hm 1.12.06		rev 1.2
	corrected failure in sequence logic.
	added init at startup to prevent from initial error after start.

hm 17.1.2007		rev 1.3
	changed output fault to status for better compatibility with other modules (ESR).
	added stop on error functionality and setup variable
	default for inputs in0..3 is true.
	renamed variable state to step

hm	17.sep 2007		rev 1.4
	replaced time() with T_PLC_MS() for compatibility reasons

*)
END_FUNCTION_BLOCK

(* POU Logic/generators/TONOF, ST *)
FUNCTION_BLOCK TONOF
VAR_INPUT
	IN : BOOL;
	T1, T2 : TIME;
END_VAR
VAR_OUTPUT
	Q : BOOL;
END_VAR
VAR
	X : TON;
	Y : TOF;
END_VAR

(*
version 1.1	17 sep 2007
programmer 	hugo
tested by		tobias

TONOF generated a TON and TOF Delay for the Input N TON (T1) and TOF (T2) can be configured separately
*)
X(IN := IN, PT := T1);
Y(in := X.Q, PT := T2);
Q := Y.Q;

(* revision history
hm	10. dec 2007	rev 1.0
	original version

*)
	
END_FUNCTION_BLOCK

(* POU Logic/memory/FIFO_16, ST *)
FUNCTION_BLOCK FIFO_16
VAR_INPUT
	Din : DWORD;
	WR : BOOL;
	E : BOOL;
	RST : BOOL;
END_VAR
VAR_OUTPUT
	Dout : DWORD := 0;
	empty : BOOL := TRUE;
	full : BOOL := FALSE;
END_VAR
VAR
	fifo : ARRAY[0..15] OF DWORD;
	NW : INT := 0;
	NR : INT := 0;
	top : INT := 15;
END_VAR

(*
	version 1.1	19. feb 2008
	programmer 	hugo
	tested by		tobias

16 Dword FIFO memory
*)
IF rst THEN
	(* asynchronous reset for the fifo *)
	NW := 0;
	NR := 0;
	Dout := 0;
	empty := TRUE;
	full := FALSE;
ELSIF WR AND E AND NOT full THEN
	(* write action *)
	fifo[NW] := Din;
	IF NW = top THEN NW := 0; ELSE NW := NW + 1; END_IF;
	full := NW = NR;
	empty := FALSE;
ELSIF NOT WR AND E AND NOT empty THEN
	(* read from stack *)
	Dout := fifo[NR];
	IF NR = top THEN NR := 0; ELSE NR := NR + 1; END_IF;
	empty := NR = NW;
	full := FALSE;
END_IF;

(* revision history
hm		4. aug. 2006	rev 1.0
	original version

hm		19. feb 2008	rev 1.1
	performance improvements

*)
END_FUNCTION_BLOCK

(* POU Logic/memory/FIFO_32, ST *)
FUNCTION_BLOCK FIFO_32
VAR_INPUT
	Din : DWORD;
	WR : BOOL;
	E : BOOL;
	RST : BOOL;
END_VAR
VAR_OUTPUT
	Dout : DWORD := 0;
	empty : BOOL := TRUE;
	full : BOOL := FALSE;
END_VAR
VAR
	fifo : ARRAY[0..31] OF DWORD;
	NW : INT := 0;
	NR : INT := 0;
	top : INT := 31;
END_VAR

(*
	version 1.1	19. feb 2008
	programmer 	hugo
	tested by		tobias

32 Dword FIFO memory
*)
IF rst THEN
	(* asynchronous reset for the fifo *)
	NW := 0;
	NR := 0;
	Dout := 0;
	empty := TRUE;
	full := FALSE;
ELSIF WR AND E AND NOT full THEN
	(* write action *)
	fifo[NW] := Din;
	IF NW = top THEN NW := 0; ELSE NW := NW + 1; END_IF;
	full := NW = NR;
	empty := FALSE;
ELSIF NOT WR AND E AND NOT empty THEN
	(* read from stack *)
	Dout := fifo[NR];
	IF NR = top THEN NR := 0; ELSE NR := NR + 1; END_IF;
	empty := NR = NW;
	full := FALSE;
END_IF;

(* revision history
hm		4. aug. 2006	rev 1.0
	original version

hm		19. feb 2008	rev 1.1
	performance improvements

*)
END_FUNCTION_BLOCK

(* POU Logic/memory/STACK_16, ST *)
FUNCTION_BLOCK STACK_16
VAR_INPUT
	Din : DWORD;
	RW : BOOL;
	E : BOOL;
	RST : BOOL;
END_VAR
VAR_OUTPUT
	Dout : DWORD := 0;
	empty : BOOL := TRUE;
	full : BOOL := FALSE;
END_VAR
VAR
	Stack : ARRAY[0..15] OF DWORD;
	N : INT := -1;
	top : INT := 15;
END_VAR

(*
	version 1.1	19 feb 2008
	programmer 	hugo
	tested by		tobias

16 Dword STACK memory
*)
IF rst THEN
	(* asynchronous reset for the fifo *)
	N := -1;
	Dout := 0;
	empty := TRUE;
	full := FALSE;
ELSIF RW AND E AND NOT full THEN
	(* write action *)
	N := N + 1;
	full := N = TOP;
	empty := FALSE;
	stack[N] := Din;
ELSIF NOT RW AND E AND NOT empty THEN
	(* read from stack *)
	Dout := stack[N];
	N := N -1;
	empty := N < 0;
	full := FALSE;
END_IF;


(* revision history
hm		4. aug. 2006	rev 1.0
	original version

hm		19. feb 2008	rev 1.1
	performance improvements

*)
END_FUNCTION_BLOCK

(* POU Logic/memory/STACK_32, ST *)
FUNCTION_BLOCK STACK_32
VAR_INPUT
	Din : DWORD;
	RW : BOOL;
	E : BOOL;
	RST : BOOL;
END_VAR
VAR_OUTPUT
	Dout : DWORD := 0;
	empty : BOOL := TRUE;
	full : BOOL := FALSE;
END_VAR
VAR
	Stack : ARRAY[0..31] OF DWORD;
	N : INT := -1;
	top : INT := 31;
END_VAR

(*
	version 1.1	19. feb 2008
	programmer 	hugo
	tested by		tobias

32 Dword STACK memory
*)
IF rst THEN
	(* asynchronous reset for the fifo *)
	N := -1;
	Dout := 0;
	empty := TRUE;
	full := FALSE;
ELSIF RW AND E AND NOT full THEN
	(* write action *)
	N := N + 1;
	full := N = TOP;
	empty := FALSE;
	stack[N] := Din;
ELSIF NOT RW AND E AND NOT empty THEN
	(* read from stack *)
	Dout := stack[N];
	N := N -1;
	empty := N < 0;
	full := FALSE;
END_IF;


(* revision history
hm		4. aug. 2006	rev 1.0
	original version

hm		19. feb 2008	rev 1.1
	performance improvements

*)
END_FUNCTION_BLOCK

(* POU Logic/Others/CRC_CHECK, ST *)
FUNCTION CRC_CHECK : BOOL
VAR_INPUT
	pt : POINTER TO ARRAY[0..32000] OF BYTE;
	size : INT;
END_VAR
VAR_INPUT CONSTANT
	Polynom_L : DWORD;
	Polynom_32 : BOOL;
END_VAR
VAR
	temp: DWORD;
END_VAR

(*
version 1.0	9 jun 2007
programmer 	hugo
tested by		tobias

CRC_CHECK checks a block of data for a crc checksum and returns true is the checksum is 0 and therfore a error free data transmission.
the CRC Polynom is specified with the config variable Polynom_L which holds the lowest 32 bits of the polynom and Polynom_33 which holds bit 33 of the Polynom.
A Polynom x4 + X + 1 is represented by 10011.
The input data is an array of byte of any size, the function is called by CRC_CHECK(ADR(array),SIZEOF(array)).

*)
temp := CRC_GEN(pt, size, polynom_L, polynom_32, 0, 0, FALSE, FALSE);
IF temp = 0 THEN CRC_CHECK := TRUE; ELSE CRC_CHECK := FALSE; END_IF;

(* typical crc polynoms

CRC-4-ITU 			x4 + x + 1 					(ITU G.704, p. 12) 	0x3 or 0xC (0x9)
CRC-5-ITU 			x5 + x4 + x2 + 1 			(ITU G.704, p. 9) 	0x15 or 0x15 (0x0B)
CRC-5-USB 			x5 + x2 + 1 				(use: USB token packets) 	0x05 or 0x14 (0x9)
CRC-6-ITU 			x6 + x + 1 					(ITU G.704, p. 3) 	0x03 or 0x30 (0x21)
CRC-7 				x7 + x3 + 1 				(use: telecom systems, MMC) 	0x09 or 0x48 (0x11)
CRC-8-ATM 			x8 + x2 + x + 1 				(use: ATM HEC) 	0x07 or 0xE0 (0xC1)
CRC-8-CCITT 		x8 + x7 + x3 + x2 + 1 		(use: 1-Wire bus) 	0x8D or 0xB1 (0x63)
CRC-8-Dallas/Maxim 	x8 + x5 + x4 + 1 			(use: 1-Wire bus) 	0x31 or 0x8C (0x19)
CRC-8 				x8 + x7 + x6 + x4 + x2 + 1 	0xD5 or 0xAB (0x57)
CRC-8-SAE J1850 	x8 + x4 + x3 + x2 + 1 		0x1D or 0xB8
CRC-10 				x10 + x9 + x5 + x4 + x + 1 	0x233 or 0x331 (0x263)
CRC-12 				x12 + x11 + x3 + x2 + x + 1 (use: telecom systems) 	0x80F or 0xF01 (0xE03)
CRC-15-CAN 			x15 + x14 + x10 + x8 + x7 + x4 + x3 + 1 	0x4599 or 0x4CD1 (0x19A3)
CRC-16-Fletcher 	Not a CRC; see Fletcher's checksum 	Used in Adler-32 A & B CRCs
CRC-16-CCITT 	x16 + x12 + x5 + 1 (XMODEM,X.25, V.41, Bluetooth, PPP, IrDA; known as "CRC-CCITT") 	0x1021 or 0x8408 (0x0811)
CRC-16-IBM 	x16 + x15 + x2 + 1 (USB, many others; also known as "CRC-16") 	0x8005 or 0xA001 (0x4003)
CRC-24-Radix-64 	x24 + x23 + x18 + x17 + x14 + x11 + x10 + x7 + x6 + x5 + x4 + x3 + x + 1 	0x864CFB or 0xDF3261 (0xBE64C3)
CRC-32-Adler 	Not a CRC; see Adler-32 	See Adler-32
CRC-32-MPEG2 	x32 + x26 + x23 + x22 + x16 + x12 + x11 + x10 + x8 + x7 + x5 + x4 + x2 + x + 1 	0x04C11DB7 or 0xEDB88320 (0xDB710641) Also used in IEEE 802.3
CRC-32-IEEE 802.3 	x32 + x26 + x23 + x22 + x16 + x12 + x11 + x10 + x8 + x7 + x5 + x4 + x2 + x + 1 (V.42) 	0x04C11DB7 or 0xEDB88320 (0xDB710641)
CRC-32C (Castagnoli) 	x32 + x28 + x27 + x26 + x25 + x23 + x22 + x20 + x19 + x18 + x14 + x13 + x11 + x10 + x9 + x8 + x6 + 1 	0x1EDC6F41 or 0x82F63B78 (0x05EC76F1)
CRC-64-ISO 	x64 + x4 + x3 + x + 1 (use: ISO 3309) 	0x000000000000001B or 0xD800000000000000 (0xB000000000000001)
CRC-64-ECMA-182 	x64 + x62 + x57 + x55 + x54 + x53 + x52 + x47 + x46 + x45 + x40 + x39 + x38 + x37 + x35 + x33 + x32 + x31 + x29 + x27 + x24 + x23 + x22 + x21 + x19 + x17 + x13 + x12 + x10 + x9 + x7 + x4 + x + 1
(as described in ECMA-182 p.63) 	0x42F0E1EBA9EA3693 or 0xC96C5795D7870F42 (0x92D8AF2BAF0E1E85)

*)

(* revision history

hm		9.6.2007	rev 1.0		original version 

*)
END_FUNCTION

(* POU Logic/Others/CRC_GEN, ST *)
FUNCTION CRC_GEN : DWORD

VAR_INPUT
	pt : POINTER TO ARRAY[0..32000] OF BYTE;
	size : INT;
END_VAR
VAR_INPUT CONSTANT
	Polynom_L : DWORD;
	Polynom_32 : BOOL;
	init: DWORD := 0;
	XOR_out : DWORD;
	rev_in : BOOL;
	rev_out : BOOL;
END_VAR
VAR
	polynom : DWORD;
	p_length : INT;
	BS : BYTE;
	data : DWORD;
	count : BYTE;
	temp : BOOL;
	step: INT;
	s4: INT;
END_VAR

(*
version 1.3	2 jan 2008
programmer 	hugo
tested by		tobias

CRC_GEN generates a CRC checksum from a block of data and returns  the checksum in a DWORD to be connected to the data for transmission.
the CRC Polynom is specified with the config variable Polynom_L which holds the lowest 32 bits of the polynom and Polynom_33 which holds bit 33 of the Polynom.
A Polynom x4 + X + 1 is represented by 10011.
The input data is an array of byte of any size, the function is called by CRC_GEN(ADR(array),SIZEOF(array)).

*)
(* check for polynom length and calculate p_length polynom will be aligned to high side of word*)
polynom := polynom_L;
IF polynom_32 THEN
	p_length := 33;
ELSE;
	p_length := 32;
	WHILE p_length > 0 AND NOT polynom.31 DO
		p_length := p_length - 1;
		Polynom := SHL(polynom,1);
	END_WHILE;
	Polynom := SHL(polynom,1);
END_IF;


(* load start code and first data byte for crc calculation *)
data := init;
IF rev_in THEN bs := reverse(pt^[0]); ELSE bs := pt^[0]; END_IF;

(* calcualte checksum *)
s4 := size + 4;
WHILE step < s4 DO
	temp := data.31;
	data := SHL(data,1);
	data.0 := BS.7;
	bs := SHL(bs,1);
	count := count + 1;
	IF count = 8 THEN
		step := step + 1;
		count := 0;
		IF step < size THEN
			IF rev_in THEN bs := reverse(pt^[step]); ELSE bs := pt^[step]; END_IF;
		END_IF;
	END_IF;
	(* check highest bit if true then xor polynom *)
	IF temp THEN data := data XOR polynom; END_IF;
END_WHILE;

(* reverse crc if necessary *)
IF rev_out THEN
	CRC_GEN.31 := data.31;
	FOR step := p_length TO 3 BY -1 DO
		data := SHL(data,1);
		CRC_GEN := SHR(CRC_GEN,1);
		CRC_GEN.31 := data.31;
	END_FOR;
ELSE
	CRC_GEN := data;
END_IF;

(* final XOR and align crc checksum to right side of dword *)
CRC_GEN := CRC_GEN XOR SHL(xor_out, 33 - p_length);
CRC_GEN := SHR(CRC_GEN,33 - p_length);


(* old code prior to rev 1.2
B1 := pt^[0];
IF size > 1 THEN B2 := pt^[1]; ELSE B2 := 0; END_IF;
IF size > 2 THEN B3 := pt^[2]; ELSE B3 := 0; END_IF;
IF size > 3 THEN B4 := pt^[3]; ELSE B4 := 0; END_IF;
IF size > 4 THEN BS := pt^[4]; ELSE BS := 0; END_IF;
data := DWord_of_Byte(B4,B3,B2,B1);

WHILE step < size DO
	temp := data.31;
	data := SHL(data,1);
	data.0 := BS.7;
	bs := SHL(bs,1);
	count := count + 1;
	IF count = 8 THEN
		step := step + 1;
		count := 0;
		IF step + 4 < size THEN bs := pt^[step+ 4]; END_IF;
	END_IF;
	(* check highest bit if true then xor polynom *)
	IF temp = TRUE THEN
		data := data XOR polynom;
	END_IF;
END_WHILE;

(* align crc checksum to right side of dword *)
CRC_GEN := SHR(data,32 - p_length +1);
*)


(* typical crc polynoms

CRC-4-ITU 			x4 + x + 1 					(ITU G.704, p. 12) 	0x3 or 0xC (0x9)
CRC-5-ITU 			x5 + x4 + x2 + 1 			(ITU G.704, p. 9) 	0x15 or 0x15 (0x0B) Bluetooth
CRC-5-USB 			x5 + x2 + 1 				(use: USB token packets) 	0x05 or 0x14 (0x9)
CRC-6-ITU 			x6 + x + 1 					(ITU G.704, p. 3) 	0x03 or 0x30 (0x21)
CRC-7 				x7 + x3 + 1 				(use: telecom systems, MMC) 	0x09 or 0x48 (0x11)
CRC-8-ATM 			x8 + x2 + x + 1 				(use: ATM HEC) 	0x07 or 0xE0 (0xC1)
CRC-8-CCITT 		x8 + x7 + x3 + x2 + 1 		(use: 1-Wire bus) 	0x8D or 0xB1 (0x63)
CRC-8-Dallas/Maxim 	x8 + x5 + x4 + 1 			(use: 1-Wire bus) 	0x31 or 0x8C (0x19)
CRC-8 				x8 + x7 + x6 + x4 + x2 + 1 	0xD5 or 0xAB (0x57)
CRC-8-SAE J1850 	x8 + x4 + x3 + x2 + 1 		0x1D or 0xB8
CRC-10 				x10 + x9 + x5 + x4 + x + 1 	0x233 or 0x331 (0x263)
CRC-12 				x12 + x11 + x3 + x2 + x + 1 (use: telecom systems) 	0x80F or 0xF01 (0xE03)
CRC-15-CAN 			x15 + x14 + x10 + x8 + x7 + x4 + x3 + 1 	0x4599 or 0x4CD1 (0x19A3)
CRC-16-Fletcher 	Not a CRC; see Fletcher's checksum 	Used in Adler-32 A & B CRCs
CRC-16-CCITT 	x16 + x12 + x5 + 1 (XMODEM,X.25, V.41, Bluetooth, PPP, IrDA; known as "CRC-CCITT") 	0x1021 or 0x8408 (0x0811)
CRC-16-IBM 	x16 + x15 + x2 + 1 (USB, many others; also known as "CRC-16") 	0x8005 or 0xA001 (0x4003)
CRC-24-Radix-64 	x24 + x23 + x18 + x17 + x14 + x11 + x10 + x7 + x6 + x5 + x4 + x3 + x + 1 	0x864CFB or 0xDF3261 (0xBE64C3)
CRC-32-Adler 	Not a CRC; see Adler-32 	See Adler-32
CRC-32-MPEG2 	x32 + x26 + x23 + x22 + x16 + x12 + x11 + x10 + x8 + x7 + x5 + x4 + x2 + x + 1 	0x04C11DB7 or 0xEDB88320 (0xDB710641) Also used in IEEE 802.3
CRC-32-IEEE 802.3 	x32 + x26 + x23 + x22 + x16 + x12 + x11 + x10 + x8 + x7 + x5 + x4 + x2 + x + 1 (V.42) 	0x04C11DB7 or 0xEDB88320 (0xDB710641)
CRC-32C (Castagnoli) 	x32 + x28 + x27 + x26 + x25 + x23 + x22 + x20 + x19 + x18 + x14 + x13 + x11 + x10 + x9 + x8 + x6 + 1 	0x1EDC6F41 or 0x82F63B78 (0x05EC76F1)
CRC-64-ISO 	x64 + x4 + x3 + x + 1 (use: ISO 3309) 	0x000000000000001B or 0xD800000000000000 (0xB000000000000001)
CRC-64-ECMA-182 	x64 + x62 + x57 + x55 + x54 + x53 + x52 + x47 + x46 + x45 + x40 + x39 + x38 + x37 + x35 + x33 + x32 + x31 + x29 + x27 + x24 + x23 + x22 + x21 + x19 + x17 + x13 + x12 + x10 + x9 + x7 + x4 + x + 1
(as described in ECMA-182 p.63) 	0x42F0E1EBA9EA3693 or 0xC96C5795D7870F42 (0x92D8AF2BAF0E1E85)

*)

(* revision history

hm		9.6.2007	rev 1.0		
	original version 

hm		11.9.2007	rev 1.1
	deleted unused variable i

hm		9. oct 2007 rev 1.2
	added init code for crc and xor_out
	added refelct in and reflect_out (rev_in und Rev_out)

hm		2. jan 2008	rev 1.3
	small changes for performance improvements
*)
END_FUNCTION

(* POU Logic/Others/matrix, ST *)
FUNCTION_BLOCK matrix
VAR_INPUT
	x1, x2, x3, x4, X5 : BOOL;
END_VAR
VAR_INPUT CONSTANT
	Release : BOOL;
END_VAR
VAR_OUTPUT
	code : BYTE;
	TP : BOOL;
	y1: BOOL := TRUE;
	y2, y3, y4 : BOOL;
END_VAR
VAR
	line : BYTE := 1;
	X : ARRAY[1..4] OF BYTE; (* scan line inputs *)
	L : ARRAY[1..4] OF BYTE; (* scan line status *)
	i: INT;
	temp: BYTE;
END_VAR

(*
version 1.2	23 dec 2007
programmer 	hugo
tested by		tobias

MATRIX is a matrix keyboard encoder for 4 rows and up to 5 columns.
matrix can send a code while a key is pressed and it sends another code while a key is released when the setup variable 'release' is set to true.
the setup variable release is false the code is only sent when the key is pressed.
the output byte holds the 5 columns in the lowest bits 0..2  and the row number in bits 4..6, while bit 7 is true for a key pressed and false for a key released.

*)
TP := FALSE;
code := 0;

(* read scan lines *)
X[line].0 := X1;
X[line].1 := X2;
X[line].2 := X3;
X[line].3 := X4;
X[line].4 := X5;

(* compare for change *)
FOR i := 1 TO 4 DO
	IF X[i] <> L[i] THEN
		(* scan line information has changed code need to be found and generated *)
		temp := x[i] XOR L[i];
		IF temp.0 THEN
			code := 1;
			code.7 := X[i].0;
			L[i].0 := X[i].0;
		ELSIF temp.1 THEN
			code := 2;
			code.7 := X[i].1;
			L[i].1 := X[i].1;
		ELSIF temp.2 THEN
			code := 3;
			code.7 := X[i].2;
			L[i].2 := X[i].2;
		ELSIF temp.3 THEN
			code := 4;
			code.7 := X[i].3;
			L[i].3 := X[i].3;
		ELSIF temp.4 THEN
			code := 5;
			code.7 := X[i].4;
			L[i].4 := X[i].4;
		END_IF;
		TP := TRUE;
		Code.4 := Line.0;
		Code.5 := Line.1;
		Code.6 := Line.2;

		(* check if release codes need to be killed *)
		IF NOT release AND code < 127 THEN
			code := 0;
			TP := 0;
		END_IF;
		EXIT;
	END_IF;
END_FOR;

(* increment scan line every cycle *)
CASE line OF
	1 :	Line := 2;
		Y1 := FALSE; Y3 := FALSE; Y4 := FALSE; Y2 := TRUE;
	2 :	Line := 3;
		Y1 := FALSE; Y2 := FALSE; Y4 := FALSE; Y3 := TRUE;
	3 :	Line := 4;
		Y1 := FALSE; Y2 := FALSE; Y3 := FALSE; Y4 := TRUE;
	4 :	Line := 1;
		Y2 := FALSE; Y3 := FALSE; Y4 := FALSE; Y1 := TRUE;
END_CASE;

(* revision history
hm		10.6.2007	rev 1.0		
	original version 


hm		11.9.2007	rev 1.1		
	deleted unused variables k and old_code

hm		23.12.2007	rev 1.2
	added exit statement in for loop instead of i:=5

*)
END_FUNCTION_BLOCK

(* POU String/CODE, ST *)
FUNCTION CODE : BYTE
VAR_INPUT
	STR : STRING;
	POS : INT;
END_VAR
VAR
	PT : POINTER TO BYTE;
END_VAR

(*
version 1.0	9. mar. 2008
programmer 	hugo
tested by		tobias

code extracts the code of a character at position POS of a string STR.

*)
IF pos < 1 OR pos > LEN(str) THEN
	CODE := 0;
	RETURN;
ELSE
	PT := ADR(STR) + INT_TO_DWORD(pos - 1);
	CODE := pt^;
END_IF;

(* revision history
hm		9. mar. 2008		rev 1.0
	original version

*)
END_FUNCTION

(* POU Mathematical/Array/_ARRAY_INIT, ST *)
FUNCTION _ARRAY_INIT : BOOL
VAR_INPUT
	pt : POINTER TO ARRAY[0..32000] OF REAL;
	size : INT;
	init : REAL;
END_VAR
VAR
	i: INT;
	stop: INT;
END_VAR


(*
version 1.2	14 nov 2007
programmer 	hugo
tested by		tobias

this function will initialize a given array with a value init.
the function needs to be called:	_array_init(adr("array"),sizeof("array"));
this function will manipulate a given array.
the function manipulates the original array, it rerturnes true when finished.
because this function works with pointers its very time efficient and it needs no extra memory.

*)
stop := SHR(size,2)-1;
FOR i := 0 TO stop DO
	pt^[i] := init;
END_FOR;

_array_init := TRUE;

(* revision History

hm 6.1.2007		rev 1.1
	change type of function to bool
	added  array_init := true to set output true.

hm	14.11.2007	rev 1.2
	changed stop calculation to be more efficient
*)
END_FUNCTION

(* POU Mathematical/Array/_ARRAY_MEDIAN, ST *)
FUNCTION _ARRAY_MEDIAN : REAL
VAR_INPUT
	pt : POINTER TO ARRAY[0..32000] OF REAL;
	size : INT;
END_VAR
VAR
	i: INT;
	stop: INT;
END_VAR

(*
version 1.4	14 nov 2007
programmer 	hugo
tested by		tobias

this function will calculate the median of a given array.
in order to do so the ariginal array is sorted and stays sorted after the function finishes
the function needs to be called:	_array_median(adr("array"),sizeof("array"));
this function will manipulate a given array.
the function will return the median of the original array.
for example [12,0,4,7,1] the median is 4 and the array after the function is called is [0,1,4,7,12]
because this function works with pointers its very time efficient and it needs no extra memory.

*)
_array_sort(pt,size);
stop := SHR(size,2)-1;
IF even(stop) THEN
	_array_median := pt^[stop/2];
ELSE
	i := SHR(stop,1);
	_array_median := (pt^[i] + pt^[i+1]) / 2;
END_IF;

(* old code
stop := (size - SIZEOF(pt)) / SIZEOF(pt);
FOR i := 0 TO stop - 1 DO
	FOR m := i + 1 TO stop DO
		IF pt^[i] > pt^[m] THEN
			temp := pt^[i];
			pt^[i] := pt^[m];
			pt^[m] := temp;
		END_IF;
	END_FOR;
END_FOR;
IF even(stop) THEN
	_array_median := pt^[stop/2];
ELSE
	i := stop/2;
	_array_median := (pt^[i] + pt^[i+1])/2;
END_IF;
*)
(* revision history
hm 	3.3.2007		rev 1.1
	corrected an error, changed the statement line 14	i := TRUNC(stop/2); to i := stop/2;

hm		22. sep 2007	rev 1.2
	changed algorithm to use _array_soft for performance reasons

hm		8. oct 2007		rev 1.3
	deleted unused variables m and temp

hm		14. nov 2007		rev 1.4
	corrected a problem with size calculation
*)
END_FUNCTION

(* POU Mathematical/Array/_ARRAY_SORT, ST *)
FUNCTION _ARRAY_SORT : BOOL
VAR_INPUT
	f : POINTER TO ARRAY[1..32000] OF REAL;
	size : INT;
END_VAR
VAR
	i: INT;
	j: INT;
	temp : REAL;
	stop : INT;
	heapsize: INT;
	popmax : REAL;
	size2: INT;
	hs2: INT;
END_VAR

(*
version 1.5	5 jan 2008
programmer 	hugo
tested by		tobias

this function will sort a given array.
the function needs to be called:	_array_sort(adr("array"),sizeof("array"));
this function will manipulate a given array.
the function will not return anything except true, it will instead manipulate the original array.
because this function works with pointers its very time efficient and it needs no extra memory.

*)
(* generate heap *)

size := SHR(size,2);
size2 := SHR(size,1);
FOR i := SIZE2  TO 1 BY -1 DO 		(* zweite Hälfte des Feldes braucht nicht betrachtet werden *)
	j:=i;
    WHILE j <= SIZE2 DO
     	stop := j * 2 + 1;               (* finde Maximum der (beiden) Söhne *)
        IF stop > SIZE THEN stop := stop - 1;
        ELSIF f^[stop-1] > f^[stop] THEN stop := stop - 1;
		END_IF;
        IF f^[j] < f^[stop] THEN   		(* ggf. tauschen *)
         	temp := f^[j];
            f^[j] := f^[stop];
            f^[stop] := temp;
        END_IF;
        j := stop;
    END_WHILE;
END_FOR;

(* heapsort *)
FOR heapsize := size TO 1 BY -1 DO
	popmax := f^[1];
	f^[1] := f^[heapsize];
   	i := 1;
	hs2 := SHR(heapsize,1);
	WHILE i <= hs2 DO	     (* letztes Element an Anfang setzen und versickern lassen *)
       	stop := i * 2 + 1;                (* finde Maximum der (beiden) Söhne *)
        	IF stop > heapsize THEN stop := stop - 1;
        	ELSIF f^[stop-1] > f^[stop] THEN stop := stop - 1;
	 	END_IF;
        	IF f^[i] < f^[stop] THEN	     (* ggf. tauschen *)
            		temp := f^[i];
            		f^[i] := f^[stop];
            		f^[stop] := temp;
        	END_IF;
        	i := stop;
    	END_WHILE;
	f^[heapsize] := popmax;
END_FOR;

_array_sort := TRUE;

(* old algorithm bubble sort used before rev 1.2
stop := (size - SIZEOF(pt)) / SIZEOF(pt);
FOR i := 0 TO stop - 1 DO
	FOR m := i + 1 TO stop DO
		IF pt^[i] > pt^[m] THEN
			temp := pt^[i];
			pt^[i] := pt^[m];
			pt^[m] := temp;
		END_IF;
	END_FOR;
END_FOR;
_array_sort := TRUE;

*)
(* revision history

hm 	6.1.2007 	rev 1.1
	changed return value to true

hm	22. sep 2007	rev 1.2
	changed sorting algorithm to heap sort for performance reasons

hm 	14. nov 2007	rev 1.3
	changed calculation of stop to be more efficient

hm	15 dec 2007		rev 1.4
	added function return true

hm	5. jan 2008		rev 1.5
	improved performance
*)
END_FUNCTION

(* POU Mathematical/Array/_ARRAY_SHUFFLE, ST *)
FUNCTION _ARRAY_SHUFFLE : BOOL
VAR_INPUT
	pt : POINTER TO ARRAY[0..32000] OF REAL;
	size : INT;
END_VAR
VAR
	temp : REAL;
	pos  : INT;
	i: INT;
	stop: INT;
END_VAR


(*
version 1.2	14 nov 2007
programmer 	kurt
tested by		hugo

this function will randomly shuffle the elements of an array
*)
stop := SHR(size,2)-1;
FOR i := 0 TO stop DO
        pos := RDM2(pos,0,stop);
        (* swap elements *)
        temp := pt^[i];
        pt^[i] := pt^[pos];
        pt^[pos] := temp;
END_FOR;

_ARRAY_SHUFFLE := TRUE;


(* revision History
hm 	4. mar 2008	rev 1.0
	original version

*)
END_FUNCTION

(* POU Mathematical/RDM2, ST *)
FUNCTION RDM2 : INT
VAR_INPUT
	last : INT;
	low : INT;
	high : INT;
END_VAR
VAR
END_VAR




(*
version 1.0	29. feb 2008
programmer 	hugo
tested by	tobias

this function calculates an integer pseudo random number
the random number will be in the range of low <= rdm2 <= high.

*)
RDM2 := TRUNC(RDM(fract(last*pi1)) * (high - low + 1)) + low;

(* revision history
hm		29. feb 2008		rev 1.0
	original version

*)
END_FUNCTION

(* POU Mathematical/Array/ARRAY_AVG, ST *)
FUNCTION ARRAY_AVG : REAL
VAR_INPUT
	pt : POINTER TO ARRAY[0..32000] OF REAL;
	size : INT;
END_VAR
VAR
	i: INT;
	stop: INT;
END_VAR

(*
version 1.1	12 dec 2007
programmer 	hugo
tested by		tobias

this function will calculate the average of a given array.
the function needs to be called:	array_avg(adr("array"),sizeof("array"));
because this function works with pointers its very time efficient and it needs no extra memory.

*)
stop := SHR(size,2)-1;
array_avg := pt^[0];
FOR i := 1 TO stop DO
	array_avg := array_avg + pt^[i];
END_FOR;
array_avg := array_avg / (stop + 1);


(* revision history
hm	2. oct 2007	rev 1.0
	original version

hm	12. dec 2007	rev 1.1
	chaged code for better performance

*)
END_FUNCTION

(* POU Mathematical/Array/ARRAY_MAX, ST *)
FUNCTION ARRAY_MAX : REAL
VAR_INPUT
	pt : POINTER TO ARRAY[0..32000] OF REAL;
	size : INT;
END_VAR
VAR
	i: INT;
	stop: INT;
END_VAR

(*
version 1.0	2 oct 2006
programmer 	hugo
tested by		tobias

this function will calculate the max value of a given array.
the function needs to be called:	array_max(adr("array"),sizeof("array"));
because this function works with pointers its very time efficient and it needs no extra memory.

*)
stop := (size -SIZEOF(pt)) / SIZEOF(pt);
array_max := pt^[0];
FOR i := 1 TO stop DO
	IF pt^[i] > array_max THEN array_max := pt^[i]; END_IF;
END_FOR;
END_FUNCTION

(* POU Mathematical/Array/ARRAY_MIN, ST *)
FUNCTION ARRAY_MIN : REAL
VAR_INPUT
	pt : POINTER TO ARRAY[0..32000] OF REAL;
	size : INT;
END_VAR
VAR
	i: INT;
	stop: INT;
END_VAR

(*
version 1.0	2 oct 2006
programmer 	hugo
tested by		tobias

this function will calculate the min value of a given array.
the function needs to be called:	array_min(adr("array"),sizeof("array"));
because this function works with pointers its very time efficient and it needs no extra memory.

*)
stop := (size - SIZEOF(pt)) / SIZEOF(pt);
array_min := pt^[0];
FOR i := 1 TO stop DO
	IF pt^[i] < array_min THEN array_min := pt^[i]; END_IF;
END_FOR;
END_FUNCTION

(* POU Mathematical/Array/ARRAY_SDV, ST *)
FUNCTION ARRAY_SDV : REAL
VAR_INPUT
	pt : POINTER TO ARRAY[0..32000] OF REAL;
	size : INT;
END_VAR
VAR
END_VAR

(*
version 1.0	1 apr 2007
programmer 	hugo
tested by		tobias

this function will calculate the standard deviation of a given array.
the function needs to be called:	array_sdv(adr("array"),sizeof("array"));
because this function works with pointers its very time efficient and it needs no extra memory.

*)
(* standard deviation is simply the square root of the variance *)

array_sdv := SQRT(array_var(pt, size));

(* revision history
hm 1.4.2007	rev 1.0
	function created
*)
END_FUNCTION

(* POU Mathematical/Array/ARRAY_VAR, ST *)
FUNCTION ARRAY_VAR : REAL
VAR_INPUT
	pt : POINTER TO ARRAY[0..32000] OF REAL;
	size : INT;
END_VAR
VAR
	avg : REAL;
	i: INT;
	stop: INT;
END_VAR

(*
version 1.1	12 dec 2007
programmer 	hugo
tested by		tobias

this function will calculate the variance of a given array.
the function needs to be called:	array_var(adr("array"),sizeof("array"));
because this function works with pointers its very time efficient and it needs no extra memory.

*)
(* at first we calualte the arithmetic average of the array *)

stop := SHR(size,2)-1;
avg := pt^[0];
FOR i := 1 TO stop DO
	avg := avg + pt^[i];
END_FOR;
avg := avg / (stop + 1);

(* in a second run we calculate the variance of the array *)

array_var := (pt^[0] - avg) * (pt^[0] - avg);
FOR i := 1 TO stop DO
	array_var := array_var + (pt^[i] - avg) * (pt^[i] - avg);
END_FOR;
array_var := array_var / stop;

(* revision history
hm 	1.4.2007	rev 1.0
	function created

hm	12.12.2007	rev 1.1
	changed code for better performance
*)
END_FUNCTION

(* POU Mathematical/Array/ARRAY_SPR, ST *)
FUNCTION ARRAY_SPR : REAL
VAR_INPUT
	pt : POINTER TO ARRAY[0..32000] OF REAL;
	size : INT;
END_VAR
VAR
	i: INT;
	stop: INT;
	array_max : REAL;
	array_min : REAL;
END_VAR

(*
version 1.0	2 oct 2006
programmer 	hugo
tested by		tobias

this function will calculate the spread of a given array.
the function needs to be called:	array_spr(adr("array"),sizeof("array"));
for example: spread of [12,0,4,1,7] is 12 - 0 = 12.
because this function works with pointers its very time efficient and it needs no extra memory.

*)
stop := (size -SIZEOF(pt)) / SIZEOF(pt);
array_min := pt^[0];
array_max := pt^[0];
FOR i := 1 TO stop DO
	IF pt^[i] > array_max THEN array_max := pt^[i];
	ELSIF pt^[i] < array_min THEN array_min := pt^[i];
	END_IF;
END_FOR;
array_spr := array_max - array_min;
END_FUNCTION

(* POU Mathematical/Array/ARRAY_SUM, ST *)
FUNCTION ARRAY_SUM : REAL
VAR_INPUT
	pt : POINTER TO ARRAY[0..32000] OF REAL;
	size : INT;
END_VAR
VAR
	i: INT;
	stop: INT;
END_VAR


(*
version 1.0	2 oct 2006
programmer 	hugo
tested by		tobias

this function will calculate the sum of a given array.
the function needs to be called:	array_sum(adr("array"),sizeof("array"));
because this function works with pointers its very time efficient and it needs no extra memory.

*)
stop := (size -SIZEOF(pt)) / SIZEOF(pt);
array_sum := pt^[0];
FOR i := 1 TO stop DO
	array_sum := array_sum + pt^[i];
END_FOR;
END_FUNCTION

(* POU Mathematical/Array/ARRAY_TREND, ST *)
FUNCTION ARRAY_TREND : REAL
VAR_INPUT
	pt : POINTER TO ARRAY[0..32000] OF REAL;
	size : INT;
END_VAR
VAR
	i: INT;
	stop: INT;
	x: REAL;
	stop2: INT;
END_VAR

(*
version 1.1	12 dec 2007
programmer 	hugo
tested by		tobias

this function will calculate the trend of a given array.
trend will calculate the avg of the first half of the array and then the avg of the second half, trend = avg2 - avg1.
for example:  [0,1,4,5,3,4,6,3] = 4 - 2.5 = 1.5
the function needs to be called:	array_trend(adr("array"),sizeof("array"));
because this function works with pointers its very time efficient and it needs no extra memory.

*)
stop := SHR(size,2)-1;
stop2 := SHR(stop,1);
FOR i := 0 TO stop2 DO x := x - pt^[i]; END_FOR;
IF even(stop) THEN
	FOR i := stop2 TO stop DO X := X + pt^[i]; END_FOR;
ELSE
	FOR i := stop2 + 1 TO stop DO X := X + pt^[i]; END_FOR;
END_IF;
array_trend := x / (stop2 + 1);

(* revision history
hm	2 oct 2007	rev 1.0
	original version

hm	12 dec 2007	rev 1.1
	changed code for better performance

*)
END_FUNCTION

(* POU Mathematical/Complex/CABS, ST *)
FUNCTION CABS : REAL
VAR_INPUT
	X : complex;
END_VAR
VAR
END_VAR

(*
version 1.0	21 feb 2008
programmer 	hugo
tested by	oscat

this function the aboslute value of a complex number

*)
CABS := HYPOT(x.re, x.im);


(* revision history
hm	21. feb 2008	rev 1.0
	original version

*)
END_FUNCTION

(* POU Mathematical/HYPOT, ST *)
FUNCTION HYPOT : REAL
VAR_INPUT
	X : REAL;
	Y : REAL;
END_VAR
VAR
END_VAR

(*
version 1.0	21 feb 2008
programmer 	hugo
tested by	oscat

this function calculates the pythagorean function

*)
HYPOT := SQRT(x*x + y*y);


(* revision history
hm	21. feb 2008	rev 1.0
	original version

*)
END_FUNCTION

(* POU Mathematical/Complex/CACOS, ST *)
FUNCTION CACOS : complex
VAR_INPUT
	X : complex;
END_VAR
VAR
	Y : complex;
END_VAR

(*
version 1.0	21 feb 2008
programmer 	hugo
tested by	oscat

this function calculates the arcus cosinus function of a complex number

*)
y := CACOSH(x);
CACOS.re := y.im;
CACOS.im := -y.re;



(* revision history
hm	21. feb 2008	rev 1.0
	original version


*)
END_FUNCTION

(* POU Mathematical/Complex/CACOSH, ST *)
FUNCTION CACOSH : complex
VAR_INPUT
	X : complex;
END_VAR
VAR
	Y : complex;
END_VAR

(*
version 1.0	21 feb 2008
programmer 	hugo
tested by	oscat

this function calculates the hyperbolic arcus cosinus function of a complex number

*)
y.re := (X.re - X.im)*(X.re + X.im) - 1.0;
y.im := 2.0 * X.re * X.im;
y    := CSQRT(y);
y.re := y.re + x.re;
y.im := y.im + x.im;
CACOSH  := CLOG(y);



(* revision history
hm	21. feb 2008	rev 1.0
	original version


*)
END_FUNCTION

(* POU Mathematical/Complex/CSQRT, ST *)
FUNCTION CSQRT : complex
VAR_INPUT
	X : complex;
END_VAR
VAR
	temp : REAL;
END_VAR

(*
version 1.0	21 feb 2008
programmer 	hugo
tested by	oscat

this function calculates the complex sqare root

*)
temp := HYPOT(x.re, x.im);
CSQRT.re :=  SQRT(0.5 * (temp + x.re));
CSQRT.im :=  sgn(x.im) * SQRT(0.5 * (temp - x.re));


(* revision history
hm	21. feb 2008	rev 1.0
	original version

*)
END_FUNCTION

(* POU Mathematical/Complex/CLOG, ST *)
FUNCTION CLOG : complex
VAR_INPUT
	X : complex;
END_VAR
VAR
END_VAR

(*
version 1.0	21 feb 2008
programmer 	hugo
tested by	oscat

this function calculates the complex natural (base e) logarithm

*)
CLOG.re := LN(HYPOT(X.re, X.im));
CLOG.im := ATAN(X.im / X.re);


(* revision history
hm	21. feb 2008	rev 1.0
	original version

*)
END_FUNCTION

(* POU Mathematical/Complex/CADD, ST *)
FUNCTION CADD : complex
VAR_INPUT
	X, Y : complex;
END_VAR
VAR
END_VAR

(*
version 1.0	21 feb 2008
programmer 	hugo
tested by	oscat

this function add two complex numbers

*)
CADD.re := x.re + y.re;
CADD.im := x.im + y.im;


(* revision history
hm	21. feb 2008	rev 1.0
	original version

*)
END_FUNCTION

(* POU Mathematical/Complex/CARG, ST *)
FUNCTION CARG : REAL
VAR_INPUT
	X : complex;
END_VAR
VAR
END_VAR

(*
version 1.0	21 feb 2008
programmer 	hugo
tested by	oscat

this function calculates the phase angle (argument) of a complex number

*)
CARG := ATAN(X.im / X.re);



(* revision history
hm	21. feb 2008	rev 1.0
	original version


*)
END_FUNCTION

(* POU Mathematical/Complex/CASIN, ST *)
FUNCTION CASIN : complex
VAR_INPUT
	X : complex;
END_VAR
VAR
	Y : complex;
END_VAR

(*
version 1.0	21 feb 2008
programmer 	hugo
tested by	oscat

this function calculates the arcus sinus function of a complex number

*)
y.re := -x.im;
y.im := x.re;
y := CASINH(y);
CASIN.re := y.im;
CASIN.im := -y.re;



(* revision history
hm	21. feb 2008	rev 1.0
	original version


*)
END_FUNCTION

(* POU Mathematical/Complex/CASINH, ST *)
FUNCTION CASINH : complex
VAR_INPUT
	X : complex;
END_VAR
VAR
	Y : complex;
END_VAR

(*
version 1.0	21 feb 2008
programmer 	hugo
tested by	oscat

this function calculates the hyperbolic arcus sinus function of a complex number

*)
y.re := (X.re - X.im)*(X.re + X.im) + 1.0;
y.im := 2.0 * X.re * X.im;
y    := CSQRT(y);
y.re := y.re + x.re;
y.im := y.im + x.im;
CASINH  := CLOG(y);



(* revision history
hm	21. feb 2008	rev 1.0
	original version


*)
END_FUNCTION

(* POU Mathematical/Complex/CATAN, ST *)
FUNCTION CATAN : complex
VAR_INPUT
	X : complex;
END_VAR
VAR
	r2: REAL;
	num, den : REAL;
END_VAR

(*
version 1.0	21 feb 2008
programmer 	hugo
tested by	oscat

this function calculates the complex arcus tangens

*)
r2 := x.re * x.re;
den := 1.0 - r2 - x.im * x.im;
CATAN.re := 0.5 * ATAN(2.0 * x.re / den);
num := x.im + 1.0;
num := r2 + num * num;
den := x.im - 1.0;
den := r2 + den * den;
CATAN.im := 0.25 * (LN(num)-LN(den));

(* revision history
hm	21. feb 2008	rev 1.0
	original version


*)
END_FUNCTION

(* POU Mathematical/Complex/CATANH, ST *)
FUNCTION CATANH : complex
VAR_INPUT
	X : complex;
END_VAR
VAR
	i2: REAL;
	num, den : REAL;
END_VAR

(*
version 1.0	21 feb 2008
programmer 	hugo
tested by	oscat

this function calculates the complex arcus hyperbolic tangens

*)
i2 := x.im * x.im;
num := 1.0 + x.re;
num := i2 + num * num;
den := 1.0 - x.re;
den := i2 + den * den;
CATANH.re := 0.25 * (LN(num) - LN(den));
den := 1 - x.re * x.re - i2;
CATANH.im := 0.5 * ATAN(2.0 * x.im / den);

(* revision history
hm	21. feb 2008	rev 1.0
	original version


*)
END_FUNCTION

(* POU Mathematical/Complex/CCON, ST *)
FUNCTION CCON : complex
VAR_INPUT
	X : complex;
END_VAR
VAR
END_VAR

(*
version 1.0	21 feb 2008
programmer 	hugo
tested by	oscat

this function calcucates the conjugation of a complex number

*)
CCON.re := x.re;
CCON.im := -x.im;


(* revision history
hm	21. feb 2008	rev 1.0
	original version

*)
END_FUNCTION

(* POU Mathematical/Complex/CCOS, ST *)
FUNCTION CCOS : complex
VAR_INPUT
	X : complex;
END_VAR
VAR
END_VAR

(*
version 1.0	21 feb 2008
programmer 	hugo
tested by	oscat

this function calculates the cosinus function of a complex number

*)
CCOS := CCOSH(CSET(-X.im, X.re));


(* revision history
hm	21. feb 2008	rev 1.0
	original version

*)
END_FUNCTION

(* POU Mathematical/Complex/CCOSH, ST *)
FUNCTION CCOSH : complex
VAR_INPUT
	X : complex;
END_VAR
VAR
END_VAR

(*
version 1.0	21 feb 2008
programmer 	hugo
tested by	oscat

this function calculates the arcus tangens function of a complex number

*)
CCOSH.re := cosH(x.re) * COS(x.im);
CCOSH.im := sinH(x.re) * SIN(x.im);


(* revision history
hm	21. feb 2008	rev 1.0
	original version

*)
END_FUNCTION

(* POU Mathematical/COSH, ST *)
FUNCTION COSH : REAL
VAR_INPUT
	X : REAL;
END_VAR
VAR
	t: REAL;
END_VAR


(*
version 1.2	5. jan 2008
programmer 	hugo
tested by		tobias

this function calculates the cos hyperbolicus

*)
T := EXP(X);
COSH := (1/T + T) * 0.5;

(* revision histroy
hm	12.1.2007	rev 1.0
	original version

hm	1.12.2007	rev 1.1
	changed code to improve performance

hm	5. jan 2008	rev 1.2
	further performance improvement
*)
END_FUNCTION

(* POU Mathematical/SINH, ST *)
FUNCTION SINH : REAL
VAR_INPUT
	X : REAL;
END_VAR
VAR
END_VAR


(*
version 1.3	11. mar 2008
programmer 	hugo
tested by	tobias

this function calculates the sin hyperbolicus

*)
IF ABS(x) < 2E-3 THEN
	SINH := X;
ELSE
	SINH := (EXP(x) - EXP(-x)) * 0.5;
END_IF;


(* revision history
hm	12.1.2007	rev 1.0
	original version

hm	1.12.2007	rev 1.1
	changed code to improve performance

hm	5. jan 2008	rev 1.2
	further performance improvement

hm	11. mar 2008	rev 1.3
	improved accuracy around 0

*)
END_FUNCTION

(* POU Mathematical/Complex/CSET, ST *)
FUNCTION CSET : complex
VAR_INPUT
	RE : REAL;
	IM : REAL;
END_VAR
VAR
END_VAR

(*
version 1.0	21 feb 2008
programmer 	hugo
tested by	oscat

this function creates a complex number from two real inputs

*)
CSET.re := RE;
CSET.im := IM;

(* revision history
hm	21. feb 2008	rev 1.0
	original version

*)
END_FUNCTION

(* POU Mathematical/Complex/CDIV, ST *)
FUNCTION CDIV : complex
VAR_INPUT
	X, Y : complex;
END_VAR
VAR
	Temp : REAL;
END_VAR

(*
version 1.0	21 feb 2008
programmer 	hugo
tested by	oscat

this function divides two complex numbers

*)
temp := Y.re * Y.re + Y.im * Y.im;
CDIV.re := (X.re * Y.re + X.im * Y.im) / temp;
CDIV.im := (X.im * Y.re - X.re * Y.im) / temp;

(* revision history
hm	21. feb 2008	rev 1.0
	original version

*)
END_FUNCTION

(* POU Mathematical/Complex/CEXP, ST *)
FUNCTION CEXP : complex
VAR_INPUT
	X : complex;
END_VAR
VAR
	Temp : REAL;
END_VAR

(*
version 1.0	21 feb 2008
programmer 	hugo
tested by	oscat

this function calculates the complex exponent

*)
temp := EXP(X.re);
CEXP.re := temp * COS(X.im);
CEXP.im := temp * SIN(X.im);


(* revision history
hm	21. feb 2008	rev 1.0
	original version

*)
END_FUNCTION

(* POU Mathematical/Complex/CINV, ST *)
FUNCTION CINV : complex
VAR_INPUT
	X : complex;
END_VAR
VAR
	temp : REAL;
END_VAR

(*
version 1.0	21 feb 2008
programmer 	hugo
tested by	oscat

this function calculates the inverse of a complex numbers (1 / X)

*)
temp := X.re * X.re + X.im * X.im;
CINV.re := X.re / temp;
CINV.im := -X.im / temp;

(* revision history
hm	21. feb 2008	rev 1.0
	original version

*)
END_FUNCTION

(* POU Mathematical/Complex/CMUL, ST *)
FUNCTION CMUL : complex
VAR_INPUT
	X, Y : complex;
END_VAR
VAR
END_VAR

(*
version 1.0	21 feb 2008
programmer 	hugo
tested by	oscat

this function multiplies two complex numbers

*)
CMUL.re := X.re * Y.re - X.im * Y.im;
CMUL.im := X.re * Y.im + X.im * Y.re;

(* revision history
hm	21. feb 2008	rev 1.0
	original version

*)
END_FUNCTION

(* POU Mathematical/Complex/CPOL, ST *)
FUNCTION CPOL : complex
VAR_INPUT
	L : REAL;
	A : REAL;
END_VAR
VAR
END_VAR

(*
version 1.0	21 feb 2008
programmer 	hugo
tested by	oscat

this function creates a complex numbers for the polar form with the inputs L (length) an A for Angle.

*)
CPOL.re := L * COS(A);
CPOL.im := L * SIN(A);


(* revision history
hm	21. feb 2008	rev 1.0
	original version

*)
END_FUNCTION

(* POU Mathematical/Complex/CPOW, ST *)
FUNCTION CPOW : complex
VAR_INPUT
	X : complex;
	Y : Complex;
END_VAR
VAR
END_VAR

(*
version 1.0	21 feb 2008
programmer 	hugo
tested by	oscat

this function calculates the complex power function x to the power of y

*)
CPOW := CEXP(CMUL(Y,CLOG(X)));


(* revision history
hm	21. feb 2008	rev 1.0
	original version

*)
END_FUNCTION

(* POU Mathematical/Complex/CSIN, ST *)
FUNCTION CSIN : complex
VAR_INPUT
	X : complex;
END_VAR
VAR
END_VAR

(*
version 1.0	21 feb 2008
programmer 	hugo
tested by	oscat

this function calculates the sinus function of a complex number

*)
CSIN.re := cosH(X.im) * SIN(X.re);
CSIN.im := sinH(X.im) * COS(X.re);


(* revision history
hm	21. feb 2008	rev 1.0
	original version

*)
END_FUNCTION

(* POU Mathematical/Complex/CSINH, ST *)
FUNCTION CSINH : complex
VAR_INPUT
	X : complex;
END_VAR
VAR
END_VAR

(*
version 1.0	21 feb 2008
programmer 	hugo
tested by	oscat

this function calculates the sinus function of a complex number

*)
CSINH.re := sinH(X.re) * COS(X.im);
CSINH.im := cosH(X.re) * SIN(X.im);


(* revision history
hm	21. feb 2008	rev 1.0
	original version

*)
END_FUNCTION

(* POU Mathematical/Complex/CSUB, ST *)
FUNCTION CSUB : complex
VAR_INPUT
	X, Y : complex;
END_VAR
VAR
END_VAR

(*
version 1.0	21 feb 2008
programmer 	hugo
tested by	oscat

this function subtracts two complex numbers

*)
CSUB.re := X.re - Y.re;
CSUB.im := X.im - Y.im;

(* revision history
hm	21. feb 2008	rev 1.0
	original version

*)
END_FUNCTION

(* POU Mathematical/Complex/CTAN, ST *)
FUNCTION CTAN : complex
VAR_INPUT
	X : complex;
END_VAR
VAR
	temp : REAL;
END_VAR

(*
version 1.0	21 feb 2008
programmer 	hugo
tested by	oscat

this function calculates the tangens function of a complex number

*)
temp := 1 / (COS(2 * x.re) + cosH( 2 * x.im));
CTAN.re := temp * SIN(2 * x.re);
CTAN.im := temp * sinH(2 * x.im);


(* revision history
hm	21. feb 2008	rev 1.0
	original version

*)
END_FUNCTION

(* POU Mathematical/Complex/CTANH, ST *)
FUNCTION CTANH : complex
VAR_INPUT
	X : complex;
END_VAR
VAR
	temp : REAL;
END_VAR

(*
version 1.0	21 feb 2008
programmer 	hugo
tested by	oscat

this function calculates the complex hyperbolictangens

*)
temp := 1 /(cosH(2 * x.re) + COS(2 * x.im));
CTANH.re := temp * sinH(2 * x.re);
CTANH.im := temp * SIN(2 * x.im);


(* revision history
hm	21. feb 2008	rev 1.0
	original version

*)
END_FUNCTION

(* POU Mathematical/functions/F_lin, ST *)
FUNCTION F_lin : REAL
VAR_INPUT
	X : REAL;
	A : REAL;
	B : REAL;
END_VAR
VAR
END_VAR

(*
version 1.0	1 sep 2006
programmer 	hugo
tested by		tobias

this function calculates the linear equation f_lin = a*x + b

*)
F_lin := A * X + B;
END_FUNCTION

(* POU Mathematical/functions/F_Lin2, ST *)
FUNCTION F_Lin2 : REAL
VAR_INPUT
	X : REAL;
	X1: REAL;
	Y1 : REAL;
	X2 : REAL;
	Y2 : REAL;
END_VAR
VAR

END_VAR

(*
version 1.0	1 jan 2007
programmer 	hugo
tested by		tobias

this function calculates the linear equation f_lin = a*x + b given by two points x1/y1 and x2/y2.

*)
F_Lin2 := (Y2 - Y1) / (X2 - X1) * X + (Y1 * X1 - Y2 * X1) / (X2 - X1) + Y1;
END_FUNCTION

(* POU Mathematical/functions/F_power, ST *)
FUNCTION F_power : REAL
VAR_INPUT
	a : REAL;
	x : REAL;
	n : REAL;
END_VAR
VAR
END_VAR

(*
version 1.0	1 sep 2006
programmer 	hugo
tested by		tobias

this function calculates the power equation f_power = a*x^n

*)
F_power := a * EXPT(X,N);
END_FUNCTION

(* POU Mathematical/functions/F_quad, ST *)
FUNCTION F_quad : REAL
VAR_INPUT
	X : REAL;
	A : REAL;
	B : REAL;
	C : REAL;
END_VAR
VAR
END_VAR

(*
version 1.0	1 sep 2006
programmer 	hugo
tested by		tobias

this function calculates the quadratic equation f_lin = a*x + b

*)
F_quad := a * X * X + B * X + C;
END_FUNCTION

(* POU Mathematical/functions/FT_avg, ST *)
FUNCTION_BLOCK FT_avg
VAR_INPUT
	in : REAL;
	en : BOOL;
	N : INT;
	rst : BOOL;
END_VAR
VAR_OUTPUT
	avg : REAL;
END_VAR
VAR
	buff : delay;
	i: INT;
	init : BOOL;
END_VAR

(*
version 1.1	7 jan 2007
programmer 	hugo
tested by		tobias

this function calculates the average over n samples from a sequential input
the input values are shifted into an N deep buffer and the avg of this buffer is diplayed at anytime on the output.
a rst will load the buffer with the current in value..

*)
(* limit n to a max of 32 because delay can do max 32 cycles *)
IF N > 32 THEN
	buff.n := 32;
ELSIF N < 0 THEN
	Buff.n := 0;
ELSE
	buff.n := N;
END_IF;

IF NOT init THEN
	FOR i := 1 TO N DO
		buff(in := in);
	END_FOR;
	avg := in;
	init := TRUE;
ELSIF rst THEN
	FOR i := 1 TO N DO
		buff(in := in);
	END_FOR;
	avg := in;
ELSIF en THEN
	buff(in := in);
	avg := avg + (in - buff.out)/N;
END_IF;

(* revision history

hm	7.1.2007	rev 1.1
	chaged rst logic to load the buffer with the actual input value instead of 0.
	added en input to allow better control of signal flow
	added init to load the buffer with in at startup to avoid rampup at beginning.
	deleted unused variable cnt.
*)
END_FUNCTION_BLOCK

(* POU Mathematical/functions/FT_min_max, ST *)
FUNCTION_BLOCK FT_min_max
VAR_INPUT
	in : REAL;
	rst : BOOL;
END_VAR
VAR_OUTPUT
	mx : REAL;
	mn : REAL;
END_VAR
VAR
	init: BOOL;
END_VAR

(*
version 1.0	1 sep 2006
programmer 	hugo
tested by		tobias

this function block stores the min and max value of an input signal.
when rst is true the mn and mx outputs are set to the in value.
when a rst is never active the function autoresets to the in value at startup.
since the input might not be present at first cycle the mn and mx are set during second cycle.

*)
IF rst OR NOT init THEN
	mn := in;
	mx := in;
	init := 1;
ELSIF in < mn THEN mn := in;
ELSIF in > mx THEN mx := in;
END_IF;
END_FUNCTION_BLOCK

(* POU Mathematical/functions/POLYNOM_INT, ST *)
FUNCTION POLYNOM_INT : REAL
VAR_INPUT
	X : REAL;
	XY : ARRAY[1..5,0..1] OF REAL;
	Pts : INT;
END_VAR
VAR
	I, J : INT;
	stop: INT;
END_VAR

(*
	version 1.2	22 feb 2008
	programmer 	oscat
	tested BY		oscat

POLYNOM_INT calculates an output based on a Polynom interpolation of up to 5 coordinates given in an array
the indut coordinates have to start at the lowest array position and must be sorted ba ascending X values.

*)
(*make sure n is bound within the array size *)
pts := MIN(pts, 5);

(* this part is only to calculate the polynom parameters, which are then stores in the Y array
	the array values, it is not needed during runtime, unless the parameters will change during runtime
	the remaining code without this setup code can be used within a function to calculate specific functions
	the content of the arrays is then used as constant values within the function *)

FOR i := 1 TO pts DO
	stop := i + 1;
   	FOR j := pts TO stop BY -1 DO
   		XY[j,1] := (XY[j,1] - XY[j-1,1]) / (XY[j,0] - XY[j-i,0]);
	END_FOR;
END_FOR;


(* this part is the actual calculation *)
POLYNOM_INT := 0;
FOR i := pts TO 1 BY -1 DO
       POLYNOM_INT := POLYNOM_INT * (X - XY[i,0]) + XY[i,1];
END_FOR;


(* revision history
hm		8. okt 2007		rev 1.0
	original version

hm		17. dec 2007	rev 1.1
	init makes no sense for a function

hm		22. feb 2008	rev 1.2
	improved performance
*)
END_FUNCTION

(* POU Mathematical/Geometry/circle_A, ST *)
FUNCTION circle_A : REAL
VAR_INPUT
	rx : REAL;
	ax : REAL;
END_VAR
VAR
END_VAR

(*
version 1.2	22. feb 2008
programmer 	hugo
tested by		tobias

circle_A calculates the Area of a circle segement if ax = 360 the whole circle is calculated


*)
circle_A := Rx * RX * 8.726646E-3 * Ax;

(* revision histroy
hm	16. oct 2007	rev 1.0
	original version

hm	4. dec 2007		rev 1.1
	changed code for better performance

hm	22. feb 2008	rev 1.2
	improved performance
*)
END_FUNCTION

(* POU Mathematical/Geometry/circle_C, ST *)
FUNCTION circle_C : REAL
VAR_INPUT
	Rx : REAL;
	Ax : REAL;
END_VAR
VAR
END_VAR

(*
version 1.1	22 feb 2008
programmer 	hugo
tested by		tobias

circle_C calculates the Circumference of a circle  if ax = 360 the whole circle is calculated

*)
circle_C := 1.7453293E-2 * Rx * Ax;

(* revision histroy
hm	16. oct 2007	rev 1.0
	original version

hm	22. feb 2008	rev 1.1
	improved performance
*)
END_FUNCTION

(* POU Mathematical/Geometry/cone_V, ST *)
FUNCTION cone_V : REAL
VAR_INPUT
	rx : REAL;
	hx : REAL;
END_VAR
VAR
END_VAR

(*
version 1.1	4 dec 2007
programmer 	hugo
tested by		tobias

cone_V calculates the Volume of a cone

*)
cone_V := 1.047197551 * RX * RX * hx;

(* revision histroy
hm	17. oct 2007	rev 1.0
	original version

hm	4. dec 2007		rev 1.1
	changed code for better performance

hm	22. feb 2008	rev 1.2
	changed code for better performance
*)
END_FUNCTION

(* POU Mathematical/Geometry/ellipse_A, ST *)
FUNCTION ellipse_A : REAL
VAR_INPUT
	R1 : REAL;
	R2 : REAL;
END_VAR
VAR
END_VAR

(*
version 1.0	16 oct 2007
programmer 	hugo
tested by		tobias

ellipse_A calculates the Area of an ellipe based on the two radians R1 and R2


*)
ellipse_A := PI1 * R1 * R2;

(* revision histroy
hm	16. oct 2007	rev 1.0
	original version

*)
END_FUNCTION

(* POU Mathematical/Geometry/ellipse_C, ST *)
FUNCTION ellipse_C : REAL
VAR_INPUT
	R1 : REAL;
	R2 : REAL;
END_VAR
VAR
END_VAR

(*
version 1.0	16 oct 2007
programmer 	hugo
tested by		tobias

ellipse_C calculates the circumference of an ellipe based on the two radians R1 and R2

*)
ellipse_C := PI1 * (3*(R1+R2) - SQRT((3*r1 + R2)*(3*r2 + r1)));

(* revision histroy
hm	16. oct 2007	rev 1.0
	original version

*)
END_FUNCTION

(* POU Mathematical/Geometry/sphere_V, ST *)
FUNCTION sphere_V : REAL
VAR_INPUT
	rx : REAL;
END_VAR
VAR
END_VAR

(*
version 1.2	22. feb 2008
programmer 	hugo
tested by		tobias

sphere_V calculates the Volume of a Sphere


*)
sphere_V := 4.188790205 * Rx * RX * RX;

(* revision histroy
hm	16. oct 2007	rev 1.0
	original version

hm	4. dec 2007		rev 1.1
	changed code for better performance

hm	22. feb 2008		rev 1.2
	changed code for better performance
*)
END_FUNCTION

(* POU Mathematical/Geometry/triangle_A, ST *)
FUNCTION triangle_A : REAL
VAR_INPUT
	S1 : REAL;
	A : REAL;
	S2 : REAL;
	S3 : REAL;
END_VAR
VAR
END_VAR

(*
version 1.1	22. feb 2008
programmer 	hugo
tested by		tobias

triangle_A calculates the Area of a triangle.
if any input is 0 it will be neglected and the are will be calculated from eiter:
two sides and an angle (s1 and S2 and the angle A1) or 3 sides.


*)
IF A = 0 THEN
	triangle_A := SQRT((s1+s2+S3) * (s1+s2-S3) * (S2+S3-S1) * (S3+S1-S2)) * 0.25;
ELSE
	triangle_A := S1 * S2 * SIN(Rad(A)) * 0.5;
END_IF;

(* revision histroy
hm	16. oct 2007	rev 1.0
	original version

hm	22. feb 2008	rev 1.1
	improved performance
*)
END_FUNCTION

(* POU Mathematical/Vektormathematik/V3_ABS, ST *)
FUNCTION V3_ABS : REAL
VAR_INPUT
	A : Vector_3;
END_VAR
VAR
END_VAR

(*
version 1.0	11 dec 2007
programmer 	hugo
tested by		tobias

this function calculates the length of a vectors in a 3 dimensional space

*)
V3_ABS := SQRT(A.X * A.X + A.Y * A.Y + A.Z * A.Z);


(* revision history
hm		11 dec 2007	rev 1.0
	original version

*)
END_FUNCTION

(* POU Mathematical/Vektormathematik/V3_ADD, ST *)
FUNCTION V3_ADD : vector_3
VAR_INPUT
	A : Vector_3;
	B : Vector_3;
END_VAR
VAR
END_VAR

(*
version 1.0	11 dec 2007
programmer 	hugo
tested by		tobias

this function adds two vectors in a 3 dimensional space

*)
V3_ADD.X := A.X + B.X;
V3_ADD.Y := A.Y + B.Y;
V3_ADD.Z := A.Z + B.Z;



(* revision history
hm		11 dec 2007	rev 1.0
	original version

*)
END_FUNCTION

(* POU Mathematical/Vektormathematik/V3_ANG, ST *)
FUNCTION V3_ANG : REAL
VAR_INPUT
	A : Vector_3;
	B : Vector_3;
END_VAR
VAR
	d : REAL;
END_VAR

(*
version 1.0	11 dec 2007
programmer 	hugo
tested by		tobias

this function calculates the angle between two vectors in a 3 dimensional space

*)
d := V3_ABS(A) * V3_ABS(B);
IF d > 0 THEN
	V3_ANG := ACOS(LIMIT(-1,V3_DPRO(A,B) / d,1));
END_IF;

(* revision history
hm		11 dec 2007	rev 1.0
	original version

*)
END_FUNCTION

(* POU Mathematical/Vektormathematik/V3_DPRO, ST *)
FUNCTION V3_DPRO : REAL
VAR_INPUT
	A : Vector_3;
	B : Vector_3;
END_VAR
VAR
END_VAR

(*
version 1.0	11 dec 2007
programmer 	hugo
tested by		tobias

this function calculates the dot product of two vectors in 3 dimensional space

*)
V3_DPRO := A.X * B.X + A.Y * B.Y + A.Z * B.Z;


(* revision history
hm		11 dec 2007	rev 1.0
	original version

*)
END_FUNCTION

(* POU Mathematical/Vektormathematik/V3_NORM, ST *)
FUNCTION V3_NORM : vector_3
VAR_INPUT
	A : Vector_3;
END_VAR
VAR
	la: REAL;
END_VAR

(*
version 1.0	11 dec 2007
programmer 	hugo
tested by		tobias

this function generates a vectors with absolute length 1 from a vector A in a 3 dimensional space

*)
la := V3_ABS(A);
IF la > 0 THEN
	V3_NORM := V3_SMUL(A,1/la);
END_IF;

(* revision history
hm		11 dec 2007	rev 1.0
	original version

*)
END_FUNCTION

(* POU Mathematical/Vektormathematik/V3_SMUL, ST *)
FUNCTION V3_SMUL : vector_3
VAR_INPUT
	A : Vector_3;
	M : REAL;
END_VAR
VAR
END_VAR

(*
version 1.0	11 dec 2007
programmer 	hugo
tested by		tobias

this function multiplies a vectors in a 3 dimensional space with a skalar M

*)
V3_SMUL.X := A.X * M;
V3_SMUL.Y := A.Y * M;
V3_SMUL.Z := A.Z * M;



(* revision history
hm		11 dec 2007	rev 1.0
	original version

*)
END_FUNCTION

(* POU Mathematical/Vektormathematik/V3_NUL, ST *)
FUNCTION V3_NUL : BOOL
VAR_INPUT
	A : Vector_3;
END_VAR
VAR
END_VAR

(*
version 1.0	12 dec 2007
programmer 	hugo
tested by		tobias

this function checks if a vectors in a null Vector

*)
V3_NUL := A.X = 0 AND A.Y = 0 AND A.Z = 0;



(* revision history
hm		12 dec 2007	rev 1.0
	original version

*)
END_FUNCTION

(* POU Mathematical/Vektormathematik/V3_PAR, ST *)
FUNCTION V3_PAR : BOOL
VAR_INPUT
	A : Vector_3;
	B : Vector_3;
END_VAR
VAR
END_VAR

(*
version 1.0	11 dec 2007
programmer 	hugo
tested by		tobias

this function checks if two vectors in a 3 dimensional space are parallel.
which means the two vectors have the same direction

*)
V3_PAR := V3_ABS(V3_XPRO(A,B)) = 0;



(* revision history
hm		11 dec 2007	rev 1.0
	original version

*)
END_FUNCTION

(* POU Mathematical/Vektormathematik/V3_XPRO, ST *)
FUNCTION V3_XPRO : vector_3
VAR_INPUT
	A : Vector_3;
	B : Vector_3;
END_VAR
VAR
END_VAR

(*
version 1.0	11 dec 2007
programmer 	hugo
tested by		tobias

this function adds two vectors in a 3 dimensional space

*)
V3_XPRO.X := A.Y * B.Z - A.Z * B.Y;
V3_XPRO.Y := A.Z * B.X - A.X * B.Z;
V3_XPRO.Z := A.X * B.Y - A.Y * B.X;



(* revision history
hm		11 dec 2007	rev 1.0
	original version

*)
END_FUNCTION

(* POU Mathematical/Vektormathematik/V3_REV, ST *)
FUNCTION V3_REV : vector_3
VAR_INPUT
	A : Vector_3;
END_VAR
VAR
END_VAR

(*
version 1.0	11 dec 2007
programmer 	hugo
tested by		tobias

this function reverses a vector in a 3 dimensional space

*)
V3_REV.X := -A.X;
V3_REV.Y := -A.Y;
V3_REV.Z := -A.Z;



(* revision history
hm		11 dec 2007	rev 1.0
	original version

*)
END_FUNCTION

(* POU Mathematical/Vektormathematik/V3_SUB, ST *)
FUNCTION V3_SUB : vector_3
VAR_INPUT
	A : Vector_3;
	B : Vector_3;
END_VAR
VAR
END_VAR

(*
version 1.0	11 dec 2007
programmer 	hugo
tested by		tobias

this function subtracts two vectors in a 3 dimensional space
V3_SUB = A - B

*)
V3_SUB.X := A.X - B.X;
V3_SUB.Y := A.Y - B.Y;
V3_SUB.Z := A.Z - B.Z;



(* revision history
hm		11 dec 2007	rev 1.0
	original version

*)
END_FUNCTION

(* POU Mathematical/Vektormathematik/V3_XANG, ST *)
FUNCTION V3_XANG : REAL
VAR_INPUT
	A : Vector_3;
END_VAR
VAR
	la: REAL;
END_VAR

(*
version 1.0	11 dec 2007
programmer 	hugo
tested by		tobias

this function calculates the angle between the X-axis and a vectors in a 3 dimensional space

*)
la := V3_ABS(a);
IF la > 0 THEN
	V3_XANG := ACOS(A.X / la);
END_IF;

(* revision history
hm		11 dec 2007	rev 1.0
	original version

*)
END_FUNCTION

(* POU Mathematical/Vektormathematik/V3_YANG, ST *)
FUNCTION V3_YANG : REAL
VAR_INPUT
	A : Vector_3;
END_VAR
VAR
	la: REAL;
END_VAR

(*
version 1.0	11 dec 2007
programmer 	hugo
tested by		tobias

this function calculates the angle between the Y-axis and a vectors in a 3 dimensional space

*)
la := V3_ABS(a);
IF la > 0 THEN
	V3_YANG := ACOS(A.Y / la);
END_IF;

(* revision history
hm		11 dec 2007	rev 1.0
	original version

*)
END_FUNCTION

(* POU Mathematical/Vektormathematik/V3_ZANG, ST *)
FUNCTION V3_ZANG : REAL
VAR_INPUT
	A : Vector_3;
END_VAR
VAR
	la: REAL;
END_VAR

(*
version 1.0	11 dec 2007
programmer 	hugo
tested by		tobias

this function calculates the angle between the Z-axis and a vectors in a 3 dimensional space

*)
la := V3_ABS(a);
IF la > 0 THEN
	V3_ZANG := ACOS(A.Z / la);
END_IF;

(* revision history
hm		11 dec 2007	rev 1.0
	original version

*)
END_FUNCTION

(* POU Mathematical/ACOSH, ST *)
FUNCTION ACOSH : REAL
VAR_INPUT
	X : REAL;
END_VAR
VAR
END_VAR


(*
version 1.1	2 dec 2007
programmer 	hugo
tested by		tobias

this function calculates the arcus cos hyperbolicus

*)
ACOSH := LN(SQRT(X * X - 1)+X);

(* revision history
hm		12 jan 2007	rev 1.0
	original version

hm		2. dec 2007	rev 1.1
	changed code for better performance

*)
END_FUNCTION

(* POU Mathematical/ACOTH, ST *)
FUNCTION ACOTH : REAL
VAR_INPUT
	X : REAL;
END_VAR
VAR
END_VAR


(*
version 1.1	5. jan 2008
programmer 	hugo
tested by		tobias

this function calculates the arcus cotangens hyperbolicus

*)
acotH := LN((x+1)/(x-1))*0.5;

(* revision history
hm		12 jan 2007	rev 1.0
	original version

hm		5. jan 2008	rev 1.1
	improved code for better performance
*)
END_FUNCTION

(* POU Mathematical/ASINH, ST *)
FUNCTION ASINH : REAL
VAR_INPUT
	X : REAL;
END_VAR
VAR
END_VAR


(*
version 1.1	2 dec 2007
programmer 	hugo
tested by		tobias

this function calculates the arcus sin hyperbolicus

*)
asinH := LN(X + SQRT(X * X + 1));

(* revision history
hm		12 jan 2007	rev 1.0
	original version

hm		2. dec 2007	rev 1.1
	changed code for better performance

*)
END_FUNCTION

(* POU Mathematical/ATANH, ST *)
FUNCTION ATANH : REAL
VAR_INPUT
	X : REAL;
END_VAR
VAR
END_VAR


(*
version 1.1	5. jan 2008
programmer 	hugo
tested by		tobias

this function calculates the arcus tangens hyperbolicus

*)
atanH := LN((1+x)/(1-x)) * 0.5;


(* revision history
hm		12 jan 2007	rev 1.0
	original version

hm		5. jan 2008	rev 1.1
	improved code for better performance
*)
END_FUNCTION

(* POU Mathematical/CEIL, ST *)
FUNCTION CEIL : INT
VAR_INPUT
	X : REAL;
END_VAR
VAR
END_VAR


(*
version 1.0	7 feb 2007
programmer 	hugo
tested by		tobias

This is a rounding function which returns the smallest possible integer which is greater or equal to X.
ceil(3.14) = 4
ceil(-3.14) = -3

*)
ceil := TRUNC(X);
IF ceil < X THEN
	ceil := ceil + 1;
END_IF;
END_FUNCTION

(* POU Mathematical/CMP, ST *)
FUNCTION CMP : BOOL
VAR_INPUT
	X,Y : REAL;
	N : INT;
END_VAR
VAR
	tmp : REAL;
END_VAR


(*
	version 1.0	12 mar 2008
	programmer 	hugo
	tested by		tobias

this function checks two inputs x and y if they are identical with the first N digits
example : cmp(3.141516,3.141517,6 is true.

*)
tmp := ABS(x);
IF tmp > 0 THEN
	tmp :=	 EXP10(FLOOR(LOG(tmp))-N+1);
ELSE
	tmp := EXP10(tmp);
END_IF;
CMP := ABS(X - Y) < tmp;


(* revision history
hm		12. mar. 2008	rev 1.0
	original version

*)
END_FUNCTION

(* POU Mathematical/FLOOR, ST *)
FUNCTION FLOOR : INT
VAR_INPUT
	X : REAL;
END_VAR
VAR
END_VAR


(*
version 1.0	7 feb 2007
programmer 	hugo
tested by		tobias

This is a rounding function which returns the biggest possible integer which is less or equal to X.
floor(3.14) = 3
floor(-3.14) = -4

*)
floor := TRUNC(X);
IF floor > X THEN
	floor := floor - 1;
END_IF;
END_FUNCTION

(* POU Mathematical/COTH, ST *)
FUNCTION COTH : REAL
VAR_INPUT
	X : REAL;
END_VAR
VAR
END_VAR


(*
version 1.3	10. mar 2008
programmer 	hugo
tested by		tobias

this function calculates the cotangens hyperbolicus

*)
IF X > 20 THEN
	cotH :=1;
ELSIF X < -20 THEN
	COTH := -1;
ELSE
	COTH := 1 + 2 / (EXP(X * 2) - 1);
END_IF;


(* revision histroy
hm		12.1.2007	rev 1.0
	original version

hm		1.12.2007	rev 1.1
	changed code to improve performance

hm		8. jan 2008	rev 1.2
	further improvement in performance

hm		10. mar 2008	rev 1.3
	extended range of valid inputs to +/- INV
	changed formula for better accuracy
*)
END_FUNCTION

(* POU Mathematical/EXPN, ST *)
FUNCTION EXPN : REAL
VAR_INPUT
	X : REAL;
	N : INT;
END_VAR
VAR
END_VAR

(*
version 1.0	 2 dec 2007
programmer 	hugo
tested by		tobias

this function calculates X to the power of N (Y = X^N) whilke N is an integer
especially on CPU's without a floating point unit this algorythm is about 30 times faster then the IEC standard EXPT() Function

*)
IF n.15 THEN
	(* N is negative *)
	N := ABS(N);
	IF N.0 THEN expn := X; ELSE expn := 1; END_IF;
	N := SHR(N,1);
	WHILE N > 0 DO
		X := X * X;
		IF N.0 THEN expn := expn * X; END_IF;
		N := SHR(N,1);
	END_WHILE;
	expn := 1 / expn;
ELSE;
	IF N.0 THEN expn := X; ELSE expn := 1; END_IF;
	N := SHR(N,1);
	WHILE N > 0 DO
		X := X * X;
		IF N.0 THEN expn := expn * X; END_IF;
		N := SHR(N,1);
	END_WHILE;
END_IF;

(* revision history
hm	4. dec 2007		rev 1.0
	original version

*)
END_FUNCTION

(* POU Mathematical/FACT, ST *)
FUNCTION FACT : DINT
VAR_INPUT
	X : INT;
END_VAR
VAR
	i: INT;
END_VAR

(*
version 1.3	10. mar. 2008
programmer 	hugo
tested by		tobias

this function calculates the factorial of x
this simple factorial only calculates factorials for inputs up to 7
if the input is negative or higher then 7 the output will be -1.

*)
IF x >= 0 AND x < 13 THEN
	FACT := 1;
	i := 2;
	WHILE i <= x DO
		FACT := FACT * i;
		i := i + 1;
	END_WHILE;
ELSE
	FACT := -1;
END_IF;

(* revision history
hm 	4.3.2007			rev 1.1
	changed a critical error where while loop was indefinite.

hm		10.12.2007		rev 1.2
	start value for i has changed to 2 for better performance

hm		10. mar 2008		rev 1.3
	changed output of fact to dint to allow bigger values
*)
END_FUNCTION

(* POU Mathematical/FIB, ST *)
FUNCTION FIB : DINT
VAR_INPUT
	X : INT;
END_VAR
VAR
	t1, t2: DINT;
END_VAR

(*
version 1.1	2 jan 2008
programmer 	hugo
tested by		tobias

this function calculates the fibonacci sequence

*)
IF FIB < 0 OR FIB > 46 THEN
	FIB := -1;
ELSIF x < 2 THEN
	FIB := X;
	RETURN;
ELSE
	(* the fibonacci number is the sum of the two suceeding fibonaci numbers *)
	(* we store the numbers alternatively in t1 and t2 depending on pt *)
	t2 := 1;
	WHILE X > 3 DO
		X := X-2;
		t1 := t1 + t2;
		t2 := t1 + t2;
	END_WHILE;
	IF X > 2 THEN t1 := t1 + t2; END_IF;
	fib := t1 + t2;
END_IF;

(* alternative code for very big numbers

IF X < 31 THEN
	fib := 0.4472136 * (expn(1.618034,X) - expn(-0.618034,X));
ELSE
	fib := 0.4472133 * expn(1.618034,X);
END_IF;

*)

(* revision history
hm		27. dec 2007	rev 1.0
	original version

hm		2. jan 2008	rev 1.1
	deleted unused variable pt

hm		10. mar 2008	rev 1.2
	changed output to dint instead of real
*)
END_FUNCTION

(* POU Mathematical/GAMMA, ST *)
FUNCTION GAMMA : REAL
VAR_INPUT
	X : REAL;
END_VAR
VAR
END_VAR

(*
version 1.0	10 dec 2007
programmer 	hugo
tested by		tobias

this function calculates the stirling function which is an approximation for the gamma function

*)
IF X >=0 THEN GAMMA := SQRT(pi2*X)*EXPT(X/E,X); END_IF;

(* revision history
hm	10.12.2007	rev 1.0
	original version

*)
END_FUNCTION

(* POU Mathematical/LANGEVIN, ST *)
FUNCTION LANGEVIN : REAL
VAR_INPUT
	X : REAL;
END_VAR
VAR
END_VAR

(*
version 1.1	11 mar 2008
programmer 	hugo
tested by		tobias

this function calculates the langevin function

*)
IF X = 0 THEN
	LANGEVIN := 0;
ELSE
	LANGEVIN := COTH(X) - 1/X;
END_IF;

(* revision history
hm	10.12.2007	rev 1.0
	original version

hm	11. mar 2008	rev 1.1
	changed formula to avoid problems when x = 0
*)
END_FUNCTION

(* POU Mathematical/MAX3, ST *)
FUNCTION MAX3 : REAL
VAR_INPUT
	in1 : REAL;
	in2 : REAL;
	in3 : REAL;
END_VAR
VAR
END_VAR

(*
version 1.0	1 jan 2007
programmer 	hugo
tested by		tobias

this function returns the highest of 3 real values

*)
IF in1 >= in2 AND in1 >= in3 THEN
	max3 := in1;
ELSIF in2 >= in1 AND in2 >= in3 THEN
	max3 := in2;
ELSE
	max3 := in3;
END_IF;
END_FUNCTION

(* POU Mathematical/MIN3, ST *)
FUNCTION MIN3 : REAL
VAR_INPUT
	in1 : REAL;
	in2 : REAL;
	in3 : REAL;
END_VAR
VAR
END_VAR

(*
version 1.0	1 jan 2007
programmer 	hugo
tested by		tobias

this function returns the lowest of 3 real values

*)
IF in1 <= in2 AND in1 <= in3 THEN
	min3 := in1;
ELSIF in2 <= in1 AND in2 <= in3 THEN
	min3 := in2;
ELSE
	min3 := in3;
END_IF;
END_FUNCTION

(* POU Mathematical/MUL_ADD, ST *)
FUNCTION MUL_ADD : REAL
VAR_INPUT
	X : REAL;
	K : REAL;
	O : REAL;
END_VAR
VAR
END_VAR

(*
version 1.1	11 nov 2007
programmer 	hugo
tested by		tobias

this function multiplies an input X with K and adds Offset O to the result.

*)
MUL_ADD := X * K + O;

(* revision history
hm	28. feb 2007
	original version

hm	11.nov 2007		rev 1.1
	deleted preset values for K and O this makes no sense for a function

*)
END_FUNCTION

(* POU Mathematical/NEG, ST *)
FUNCTION NEG : INT
VAR_INPUT
	in : INT;
END_VAR
VAR
	X : WORD := 2#1111_1111_1111_1111;
END_VAR

(*
version 1.0	11 nov 2007
programmer 	hugo
tested by		tobias

this function return the value of in multiplied by -1

*)
NEG := WORD_TO_INT(INT_TO_WORD(in - 1) XOR X);

(* revision history
hm 11.11.2007	rev 1.0
	original version

*)
END_FUNCTION

(* POU Mathematical/RDMDW, ST *)
FUNCTION RDMDW : DWORD
VAR_INPUT
	last : DWORD;
END_VAR
VAR
	RX: REAL;
	M: REAL;
END_VAR




(*
version 1.0	14. mar 2008
programmer 	hugo
tested by		tobias

this function calculates a DWORD pseudo random number.

*)
M := BIT_COUNT(last);
RX := RDM(FRACT(M*pi1));
RDMDW := SHL(REAL_TO_DWORD(rx*65535),16);
RX := RDM(FRACT(M*e));
RDMDW := RDMDW OR (REAL_TO_DWORD(rx*65535) AND 16#0000FFFF);



(* revision history
hm		14. mar 2008		rev 1.0
	original version

*)
END_FUNCTION

(* POU Mathematical/RND, ST *)
FUNCTION RND : REAL
VAR_INPUT
	X : REAL;
	N : INT;
END_VAR
VAR
	M : REAL;
	LX : INT;
END_VAR

(*
version 1.0	11. mar 2008
programmer 	hugo
tested by	tobias

this function rounds a real down to n digits total.
round(3.1415,2) = 3.1

*)
IF X = 0 THEN
	RND := 0;
ELSE
      LX := CEIL(LOG(ABS(X)));
      M := EXPN(10,N-LX);
      RND := DINT_TO_REAL(REAL_TO_DINT(X * M)) / M;
END_IF;



(* revision history
hm	11. mar 2008	rev 1.0
	original version

*)
END_FUNCTION

(* POU Mathematical/ROUND, ST *)
FUNCTION ROUND : REAL
VAR_INPUT
	in : REAL;
	N : INT;
END_VAR
VAR
	X: REAL;
END_VAR

(*
version 1.3	11. mar 2008
programmer 	hugo
tested by	tobias

this function rounds a real down to n digits behind the comma.
round(3.1415,1) = 3.1

*)
IF N < 4 THEN
	IF N < 2 THEN
		IF N = 0 THEN X := 1; ELSE X := 10; END_IF;
	ELSE
		IF N = 2 THEN X := 100; ELSE X := 1000; END_IF;
	END_IF;
ELSE
	IF N < 6 THEN
		IF N = 4 THEN X := 10000; ELSE X := 100000; END_IF;
	ELSE
		IF N = 6 THEN X := 1000000; ELSE X := 10000000; END_IF;
	END_IF;
END_IF;

ROUND := REAL_TO_DINT(in * X) / X;
(*
IF in >= 0 THEN
	ROUND := TRUNC(in * X + 0.5) / X;
ELSE
	ROUND := TRUNC(in * X - 0.5) / X;
END_IF;
*)

(* revision history
hm	1. sep 2006	rev 1.0
	original version

hm	2. dec 2007	rev 1.1
	changed code for better performance

hm	8. jan 2008	rev 1.2
	further improvement in performance

hm 11. mar. 2008	rev 1.3
	corrected an error with negative numbers
	use real_to_dint instead of trunc

*)
END_FUNCTION

(* POU Mathematical/SIGMOID, ST *)
FUNCTION SIGMOID : REAL
VAR_INPUT
	X : REAL;
END_VAR
VAR
END_VAR

(*
version 1.1	11.  mar 2008
programmer 	hugo
tested by	tobias

this function calculates the sigmoid function

*)
IF X > 20 THEN
	SIGMOID := 1;
ELSIF x < -85 THEN
	SIGMOID := 0;
ELSE
	SIGMOID := 1 / (1 + EXP(-X));
END_IF;

(* revision history
hm		10.12.2007		rev 1.0
	original version

hm		11. mar. 2008		rev 1.1
	extended range of valid inputs to +inv / -inv

*)
END_FUNCTION

(* POU Mathematical/SIGN_I, ST *)
FUNCTION SIGN_I : BOOL
VAR_INPUT
	in : INT;
END_VAR
VAR
END_VAR

(*
version 1.2	1 dec 2007
programmer 	hugo
tested by	tobias

this function return true if the integer input is negative

*)
sign_I := in.15;

(* revision history
hm 3.3.2007	rev 1.1
	changed method of function for better compatibility to other systems

hm	1.12.2007	rev 1.2
	changed code to improve performance
*)
END_FUNCTION

(* POU Mathematical/SINC, ST *)
FUNCTION SINC : REAL
VAR_INPUT
	X : REAL;
END_VAR
VAR
END_VAR


(*
version 1.0	11. mar 2008
programmer 	hugo
tested by		tobias

this function calculates the sinc function.

*)
IF X = 0 THEN
	SINC := 1;
ELSE
	SINC := SIN(x) / x;
END_IF;


(* revision histroy
hm	11. mar. 2008
	original version

hm	1.12.2007	rev 1.1
	changed code to improove performance

*)
END_FUNCTION

(* POU Mathematical/SQRTN, ST *)
FUNCTION SQRTN : REAL
VAR_INPUT
	X : REAL;
	N : INT;
END_VAR
VAR
END_VAR

(*
version 1.2	11. mar 2008
programmer 	hugo
tested by	tobias

this function calculates the nth root function of X according to the formula sqrtn = x^(1/n).

*)
IF N > 0 THEN
	(*	sqrtn := EXPT(x, 1.0 / INT_TO_REAL(n)); old code in rev 1.0 *)
	SQRTN := EXP(LN(x)/n);
ELSE
	SQRTN := 0;
END_IF;


(* revision history
hm		12 jan 2007	rev 1.0
	original version

hm		2. dec 2007	rev 1.1
	changed code for better performance

hm		11. mar 2008	rev 1.2
	added result 0 for compatibility reasons
*)
END_FUNCTION

(* POU Mathematical/TANH, ST *)
FUNCTION TANH : REAL
VAR_INPUT
	X : REAL;
END_VAR
VAR
END_VAR


(*
version 1.2	10. mar 2008
programmer 	hugo
tested by	tobias

this function calculates the tangens hyperbolicus

*)
IF X > 20 THEN
	tanH := 1;
ELSIF X < -20 THEN
	tanH := -1;
ELSE
	tanH := 1 - 2 / (EXP(2 * x) + 1);
END_IF;

(* revision hisdtory
hm		12.1.2007		rev 1.0
	original version

hm		1.12.2007		rev 1.1
	changed code to improve performance

hm		10. mar 2008	rev 1.2
	corrected an error in formula
	extended range of valid inputs to +/- INV
*)
END_FUNCTION

(* POU Mathematical/WINDOW, ST *)
FUNCTION WINDOW : BOOL
VAR_INPUT
	low : REAL;
	in : REAL;
	high : REAL;
END_VAR
VAR
END_VAR

(*
	version 1.1	22 jan 2007
	programmer 	hugo
	tested BY	tobias

this checks a signal if the signal is between the upper and lower limit
*)
window := in < high AND in > low;


(* revision history
hm	22.1.2007	rev 1.1
	changed the order of inputs to low, in, high

*)
END_FUNCTION

(* POU Mathematical/WINDOW2, ST *)
FUNCTION WINDOW2 : BOOL
VAR_INPUT
	low : REAL;
	in : REAL;
	high : REAL;
END_VAR
VAR
END_VAR

(*
	version 1.0	31 oct 2007
	programmer 	hugo
	tested BY	tobias

this checks a signal if the signal is between the upper and lower limit including the two limits
*)
WINDOW2 := in <= high AND in >= low;


(* revision history
hm	31.10.2007	rev 1.0
	original version

*)
END_FUNCTION

(* POU Network/IP4_CHECK, ST *)
FUNCTION IP4_CHECK : BOOL
VAR_INPUT
	NIP : DWORD;
	LIP : DWORD;
	SM : DWORD;
END_VAR
VAR
END_VAR

(*
version 1.0	4. mar 2008
programmer 	hugo
tested by		oscat

IP4_CHECK testet ob eine Network IP und Local_IP im selben Subnet sind.

*)
IP4_CHECK := (NIP AND sm) = (LIP AND SM);


(* revision history
hm		4. mar 2008	rev 1.0
	original version

*)
END_FUNCTION

(* POU Network/IP4_DECODE, ST *)
FUNCTION IP4_DECODE : DWORD
VAR_INPUT
	str : STRING;
END_VAR
VAR
	d1, d2, d3, d4 : INT;
	s1, s2, s3, s4 : STRING(3);
END_VAR

(*
version 1.0	29. feb 2008
programmer 		kurt
tested by		hugo

IP4_DECODE testet ob ein string eine gültige IPv4 Adresse enthält und gibt die 4 Bytes der IP Adresse als DWORD zurück.

*)
IP4_DECODE := 0;
(* check wheather 3 dots are present *)
IF COUNT_CHAR(str,46) <> 3 THEN RETURN; END_IF;
(* store the positions of the 3 dots *)
d1 := FINDP(str,'.',1);
d2 := FINDP(str,'.',d1+1);
d3 := FINDP(str,'.',d2+1);
IF d1 > 4 OR d2 - d1 > 4 OR d3 - d2 > 4 THEN RETURN; END_IF;
(* store the 3 strings between the dots in d1 .. d4 *)
s1 := LEFT(str,d1-1);
s2 := MID(str,d2-d1-1,d1+1);
s3 := MID(str,d3-d2-1,d2+1);
s4 := RIGHT(str,LEN(str)-d3);
(* check if the 3 strings are numbers only *)
IF NOT IS_NUM(s1) OR NOT IS_NUM(s2) OR NOT IS_NUM(s3) OR NOT IS_NUM(s4) THEN RETURN; END_IF;
(* convert the 4 numbers and check range 0..255 *)
d1 := STRING_TO_INT(s1);
d2 := STRING_TO_INT(s2);
d3 := STRING_TO_INT(s3);
d4 := STRING_TO_INT(s4);
(* check range of numbers *)
IF d1 > 255 OR d2 > 255 OR d3 > 255 OR d4 > 255 THEN RETURN; END_IF;
(* convert to output *)
IP4_DECODE := SHL(INT_TO_DWORD(d1),24) OR SHL(INT_TO_DWORD(d2),16) OR SHL(INT_TO_DWORD(d3),8) OR INT_TO_DWORD(d4);



(* revision history
hm		29. feb 2008	rev 1.0
	original version

*)
END_FUNCTION

(* POU String/COUNT_CHAR, ST *)
FUNCTION COUNT_CHAR : INT
VAR_INPUT
	str : STRING;
	chr : BYTE;
END_VAR
VAR
	l: INT;
	pt : POINTER TO BYTE;
	pos: INT;
END_VAR


(*
version 1.0	29. feb 2008
programmer 		kurt
tested by		hugo

COUNT_CHAR how often a character CHAR occurs within a string STR.

*)
PT := ADR(str);
l := LEN(str);
COUNT_CHAR := 0;
FOR pos := 1 TO l DO
	IF pt^ = CHR THEN COUNT_CHAR := COUNT_CHAR + 1; END_IF;
    PT := PT + 1;
END_FOR;


(* revision history
hm		29. feb 2008	rev 1.0
	original version

*)
END_FUNCTION

(* POU String/CHR, ST *)
FUNCTION CHR : STRING
VAR_INPUT
	C : BYTE;
END_VAR
VAR
	PT : POINTER TO BYTE;
END_VAR

(*
version 1.1	4. feb 2008
programmer 	hugo
tested by		tobias

CHR creates a character from a byte input and stuffs it in a one character length string.

*)
PT := ADR(CHR);
PT^ := C;
pt := pt + 1;
pt^ := 0;

(* revision history
hm		16 jan 2007		rev 1.0
	original version

hm		4. feb. 2008		rev 1.1
	return string would not be terminated properly
*)
END_FUNCTION

(* POU String/FINDP, ST *)
FUNCTION FINDP : INT
VAR_INPUT
	str : STRING;
	src : STRING;
	pos: INT;
END_VAR
VAR
	i: INT;
	ls: INT;
	lx: INT;
	stp: INT;
END_VAR

(*
version 1.1	29. feb 2009
programmer 	hugo
tested by		tobias

the function findP searches a string str for the occurence of src beginning at the position pos.

*)
ls := LEN(str);
lx := LEN(src);
IF ls < lx OR lx = 0 THEN RETURN; END_IF;
stp := ls - lx + 1;
FOR i := MAX(pos,1) TO stp DO
	IF MID(str,lx,i) = src THEN
		FINDP := i;
		RETURN;
	END_IF;
END_FOR;
FINDP := 0;

(* revision histroy
hm		4. feb. 2008	rev 1.0
	original release

hm		29. feb 2008	rev 1.1
	ADDED MAX(pos,1) in loop initialization

*)	
END_FUNCTION

(* POU String/IS_NUM, ST *)
FUNCTION IS_NUM : BOOL
VAR_INPUT
	str : STRING;
END_VAR
VAR
	L : INT;
	pt : POINTER TO BYTE;
	pos: INT;
END_VAR

(*
version 1.0	29. feb 2008
programmer 		kurt
tested by		hugo

IS_NUM testet ob in einem string nur Zahlen 0..9 vorkommen.

*)
PT := ADR(str);
L := LEN(str);
FOR pos := 1 TO L DO
	IF NOT (ISC_NUM(pt^)) THEN
		IS_NUM := FALSE;
		RETURN;
	END_IF;
    	PT := PT + 1;
END_FOR;
IS_NUM := L > 0;


(* revision history
hm		29. feb 2008	rev 1.0
	original version

*)
END_FUNCTION

(* POU String/ISC_NUM, ST *)
FUNCTION ISC_NUM : BOOL
VAR_INPUT
	IN : BYTE;
END_VAR
VAR
END_VAR

(*
version 1.0	6. mar 2008
programmer 	oscat
tested by		hugo

ISC_NUM checks if a character is 0..9.

*)
ISC_NUM := IN > 47 AND IN < 58;

(* revision history
hm		6. mar. 2008	rev 1.0
	original version

*)
END_FUNCTION

(* POU Network/IS_IP4, ST *)
FUNCTION IS_IP4 : BOOL
VAR_INPUT
	str : STRING;
END_VAR
VAR
END_VAR

(*
version 1.0	1. mar 2008
programmer 		kurt
tested by		hugo

IS_IP4 testet ob ein string eine gültige IPv4 Adresse enthält.

*)
IS_IP4 := IP4_DECODE(str) > 0;


(* revision history
hm		1. mar 2008	rev 1.0
	original version

*)
END_FUNCTION

(* POU Other/ESR_collect, ST *)
FUNCTION_BLOCK ESR_collect
VAR_INPUT
	ESR_0, ESR_1, ESR_2, ESR_3, ESR_4, ESR_5, ESR_6, ESR_7 : ARRAY [0..3] OF esr_data;
	RST : BOOL;
END_VAR
VAR_OUTPUT
	ESR_OUT : ARRAY[0..63] OF esr_data;
	pos : INT;
END_VAR
VAR CONSTANT
	max_in : INT := 3; (* maximum element of input variable *)
	max_out : INT := 63; (* maximum element of output array *)
END_VAR
VAR
	cnt : INT;
END_VAR

(*
version 1.0	26 jan 2007
programmer 	hugo
tested by		tobias

ESR_collect collects esr data from up to 8 esr_mon modules and stroes them in an output array.
the output pos will display the position of the last element in the array.
if the array will be full, the oldest element is overwritten.

*)
IF rst THEN
	pos := 0;
	FOR cnt := 0 TO 63 DO
		esr_out[cnt].typ := 0;
		esr_out[cnt].adress := '';
		esr_out[cnt].DS := DT#1970-1-1-00:00;
		esr_out[cnt].TS := T#0ms;
		esr_out[cnt].data[0] := 0;
		esr_out[cnt].data[1] := 0;
		esr_out[cnt].data[2] := 0;
		esr_out[cnt].data[3] := 0;
		esr_out[cnt].data[4] := 0;
		esr_out[cnt].data[5] := 0;
		esr_out[cnt].data[6] := 0;
		esr_out[cnt].data[7] := 0;
	END_FOR;
ELSE
	FOR cnt := 0 TO max_in DO
		IF esr_0[cnt].typ > 0 THEN
			esr_out[pos] := esr_0[cnt];
			pos := pos + 1;
			IF pos > max_out THEN pos := 0; END_IF;
		END_IF;
	END_FOR;
	FOR cnt := 0 TO max_in DO
		IF esr_1[cnt].typ > 0 THEN
			esr_out[pos] := esr_1[cnt];
			pos := pos + 1;
			IF pos > max_out THEN pos := 0; END_IF;
		END_IF;
	END_FOR;
	FOR cnt := 0 TO max_in DO
		IF esr_2[cnt].typ > 0 THEN
			esr_out[pos] := esr_2[cnt];
			pos := pos + 1;
			IF pos > max_out THEN pos := 0; END_IF;
		END_IF;
	END_FOR;
	FOR cnt := 0 TO max_in DO
		IF esr_3[cnt].typ > 0 THEN
			esr_out[pos] := esr_3[cnt];
			pos := pos + 1;
			IF pos > max_out THEN pos := 0; END_IF;
		END_IF;
	END_FOR;
	FOR cnt := 0 TO max_in DO
		IF esr_4[cnt].typ > 0 THEN
			esr_out[pos] := esr_4[cnt];
			pos := pos + 1;
			IF pos > max_out THEN pos := 0; END_IF;
		END_IF;
	END_FOR;
	FOR cnt := 0 TO max_in DO
		IF esr_5[cnt].typ > 0 THEN
			esr_out[pos] := esr_5[cnt];
			pos := pos + 1;
			IF pos > max_out THEN pos := 0; END_IF;
		END_IF;
	END_FOR;
	FOR cnt := 0 TO max_in DO
		IF esr_6[cnt].typ > 0 THEN
			esr_out[pos] := esr_6[cnt];
			pos := pos + 1;
			IF pos > max_out THEN pos := 0; END_IF;
		END_IF;
	END_FOR;
	FOR cnt := 0 TO max_in DO
		IF esr_7[cnt].typ > 0 THEN
			esr_out[pos] := esr_7[cnt];
			pos := pos + 1;
			IF pos > max_out THEN pos := 0; END_IF;
		END_IF;
	END_FOR;
END_IF;

(* revision history
hm	26.jan 2007		rev 1.0
	original version

hm	8. dec 2007		rev 1.1
	added reset input

*)
END_FUNCTION_BLOCK

(* POU Other/ESR_MON_B8, ST *)
FUNCTION_BLOCK ESR_MON_B8
VAR_INPUT
	s0, s1, s2, s3, s4, s5, s6, s7 : BOOL;
	DT_in : DT;
END_VAR
VAR_INPUT CONSTANT
	a0, a1, a2, a3, a4, a5, a6, a7 : STRING(10);
END_VAR
VAR_OUTPUT
	ESR_Out: ARRAY [0..3] OF esr_data;
	ESR_Flag : BOOL;
END_VAR
VAR
	x0, x1, x2, x3, x4, x5, x6, x7 : BOOL;
	tx: TIME;
	cnt : INT;
END_VAR

(*
version 1.1	17 sep 2007
programmer 	hugo
tested by		tobias

ESR_mon_B8 monitores up to 8 binary inputs and reports changes with time stamd and adress label.
the module checks 8 inputs for a change and reports all changes with time and adress stamp to the output.
4 events maximum can be collected at once within the same cycle

*)
(* read system timer *)
tx := DWORD_TO_TIME(T_PLC_MS());

ESR_Flag := FALSE;
esr_out[3].typ := 0;
esr_out[2].typ := 0;
esr_out[1].typ := 0;
esr_out[0].typ := 0;
cnt := 0;

(* check if inputs have chaged and fill buffer *)
IF s0 <> X0 THEN
	IF s0 THEN esr_out[cnt].typ := 11; ELSE 	esr_out[cnt].typ := 10; END_IF;
	esr_out[cnt].adress := a0;
	esr_out[cnt].DS := DT_in;
	esr_out[cnt].TS := TX;
	X0 := S0;
	cnt := cnt + 1;
	esr_flag := TRUE;
END_IF;
IF s1 <> X1 THEN
	IF s1 THEN esr_out[cnt].typ := 11; ELSE 	esr_out[cnt].typ := 10; END_IF;
	esr_out[cnt].adress := a1;
	esr_out[cnt].DS := DT_in;
	esr_out[cnt].TS := TX;
	X1 := S1;
	cnt := cnt + 1;
	esr_flag := TRUE;
END_IF;
IF s2 <> X2 THEN
	IF s2 THEN esr_out[cnt].typ := 11; ELSE 	esr_out[cnt].typ := 10; END_IF;
	esr_out[cnt].adress := a2;
	esr_out[cnt].DS := DT_in;
	esr_out[cnt].TS := TX;
	X2 := S2;
	cnt := cnt + 1;
	esr_flag := TRUE;
END_IF;
IF s3 <> X3 THEN
	IF s3 THEN esr_out[cnt].typ := 11; ELSE 	esr_out[cnt].typ := 10; END_IF;
	esr_out[cnt].adress := a3;
	esr_out[cnt].DS := DT_in;
	esr_out[cnt].TS := TX;
	X3 := S3;
	cnt := cnt + 1;
	esr_flag := TRUE;
END_IF;
IF s4 <> X4 AND cnt < 4 THEN
	IF s4 THEN esr_out[cnt].typ := 11; ELSE 	esr_out[cnt].typ := 10; END_IF;
	esr_out[cnt].adress := a4;
	esr_out[cnt].DS := DT_in;
	esr_out[cnt].TS := TX;
	X4 := S4;
	cnt := cnt + 1;
	esr_flag := TRUE;
END_IF;
IF s5 <> X5  AND cnt < 4 THEN
	IF s5 THEN esr_out[cnt].typ := 11; ELSE 	esr_out[cnt].typ := 10; END_IF;
	esr_out[cnt].adress := a5;
	esr_out[cnt].DS := DT_in;
	esr_out[cnt].TS := TX;
	X5 := S5;
	cnt := cnt + 1;
	esr_flag := TRUE;
END_IF;
IF s6 <> X6  AND cnt < 4 THEN
	IF s6 THEN esr_out[cnt].typ := 11; ELSE 	esr_out[cnt].typ := 10; END_IF;
	esr_out[cnt].adress := a6;
	esr_out[cnt].DS := DT_in;
	esr_out[cnt].TS := TX;
	X6 := S6;
	cnt := cnt + 1;
	esr_flag := TRUE;
END_IF;
IF s7 <> X7  AND cnt < 4 THEN
	IF s7 THEN esr_out[cnt].typ := 11; ELSE 	esr_out[cnt].typ := 10; END_IF;
	esr_out[cnt].adress := a7;
	esr_out[cnt].DS := DT_in;
	esr_out[cnt].TS := TX;
	X7 := S7;
	cnt := cnt + 1;
	esr_flag := TRUE;
END_IF;

(* revision history
hm	26. jan 2007		rev 1.0
	original version

hm	17. sep 2007	rev 1.1
	replaced time() with T_PLC_MS() for compatibility reasons
	
*)
END_FUNCTION_BLOCK

(* POU Other/ESR_MON_R4, ST *)
FUNCTION_BLOCK ESR_MON_R4
VAR_INPUT
	R0, R1, R2, R3 : REAL;
	DT_in : DT;
END_VAR
VAR_INPUT CONSTANT
	a0, a1, a2, a3 : STRING(10);
	s0, s1, s2, s3 : REAL;
END_VAR
VAR_OUTPUT
	ESR_Out: ARRAY [0..3] OF esr_data;
	ESR_Flag : BOOL;
END_VAR
VAR
	p0, p1, p2, p3 : POINTER TO DWORD;
	x0, x1, x2, x3 : REAL;
	tx: TIME;
	cnt : INT;
END_VAR

(*
version 1.2 8 dec 2007
programmer 	hugo
tested by		tobias

ESR_mon_R4 monitores up to 4 Real inputs and reports changes with time stamd and adress label.
the module checks 4 inputs for a change of more than the specified sensitivity S and reports all changes with time and adress stamp to the output.

*)
(* read system timer *)
tx := DWORD_TO_TIME(T_PLC_MS());
P0 := ADR(R0);
P1 := ADR(R1);
P2 := ADR(R2);
P3 := ADR(R3);

ESR_Flag := FALSE;
esr_out[3].typ := 0;
esr_out[2].typ := 0;
esr_out[1].typ := 0;
esr_out[0].typ := 0;
cnt := 0;

(* check if inputs have chaged and fill buffer *)
IF differ(R0,  X0, S0) THEN
	esr_out[cnt].typ := 20;
	esr_out[cnt].adress := a0;
	esr_out[cnt].DS := DT_in;
	esr_out[cnt].TS := TX;
	esr_out[cnt].data[0] := Byte_of_Dword(REAL_TO_DWORD(P0^),0);
	esr_out[cnt].data[1] := Byte_of_Dword(REAL_TO_DWORD(P0^),1);
	esr_out[cnt].data[2] := Byte_of_Dword(REAL_TO_DWORD(P0^),2);
	esr_out[cnt].data[3] := Byte_of_Dword(REAL_TO_DWORD(P0^),3);
	X0 := R0;
	cnt := cnt + 1;
	esr_flag := TRUE;
END_IF;
IF differ(R1,  X1, S1) THEN
	esr_out[cnt].typ := 20;
	esr_out[cnt].adress := a1;
	esr_out[cnt].DS := DT_in;
	esr_out[cnt].TS := TX;
	esr_out[cnt].data[0] := Byte_of_Dword(REAL_TO_DWORD(P1^),0);
	esr_out[cnt].data[1] := Byte_of_Dword(REAL_TO_DWORD(P1^),1);
	esr_out[cnt].data[2] := Byte_of_Dword(REAL_TO_DWORD(P1^),2);
	esr_out[cnt].data[3] := Byte_of_Dword(REAL_TO_DWORD(P1^),3);
	X1 := R1;
	cnt := cnt + 1;
	esr_flag := TRUE;
END_IF;
IF differ(R2,  X2, S2) THEN
	esr_out[cnt].typ := 20;
	esr_out[cnt].adress := a2;
	esr_out[cnt].DS := DT_in;
	esr_out[cnt].TS := TX;
	esr_out[cnt].data[0] := Byte_of_Dword(REAL_TO_DWORD(P2^),0);
	esr_out[cnt].data[1] := Byte_of_Dword(REAL_TO_DWORD(P2^),1);
	esr_out[cnt].data[2] := Byte_of_Dword(REAL_TO_DWORD(P2^),2);
	esr_out[cnt].data[3] := Byte_of_Dword(REAL_TO_DWORD(P2^),3);
	X2 := R2;
	cnt := cnt + 1;
	esr_flag := TRUE;
END_IF;
IF differ(R3,  X3, S3) THEN
	esr_out[cnt].typ := 20;
	esr_out[cnt].adress := a3;
	esr_out[cnt].DS := DT_in;
	esr_out[cnt].TS := TX;
	esr_out[cnt].data[0] := Byte_of_Dword(REAL_TO_DWORD(P3^),0);
	esr_out[cnt].data[1] := Byte_of_Dword(REAL_TO_DWORD(P3^),1);
	esr_out[cnt].data[2] := Byte_of_Dword(REAL_TO_DWORD(P3^),2);
	esr_out[cnt].data[3] := Byte_of_Dword(REAL_TO_DWORD(P3^),3);
	X3 := R3;
	cnt := cnt + 1;
	esr_flag := TRUE;
END_IF;


(* revision history
hm	26. jan 2007	rev 1.0
	original version

hm	17. sep 2007	rev 1.1
	replaced time() with T_PLC_MS() for compatibility reasons

hm	8 dec 2007		rev 1.2
	corrected an error while esr typ would not be set
*)
END_FUNCTION_BLOCK

(* POU Other/ESR_MON_X8, ST *)
FUNCTION_BLOCK ESR_MON_X8
VAR_INPUT
	s0, s1, s2, s3, s4, s5, s6, s7 : BYTE;
	DT_in : DT;
	Mode : BYTE := 3;
END_VAR
VAR_INPUT CONSTANT
	a0, a1, a2, a3, a4, a5, a6, a7 : STRING(10);
END_VAR
VAR_OUTPUT
	ESR_Out: ARRAY [0..3] OF esr_data;
	ESR_Flag : BOOL;
END_VAR
VAR
	x0, x1, x2, x3, x4, x5, x6, x7 : BYTE;
	tx: TIME;
	cnt : INT;
END_VAR

(*
version 1.1	17 sep 2007
programmer 	hugo
tested by		tobias

ESR_MON_X8 is a status and error collector.
the module checks 8 status inputs for a change and reports up to 4 input changes with time and adress stamp to the output.
the mode can be 
1 for error only
2 for error and status
3 for error, status and debug
the adress label of the 8 inputs can be configured individually.
*)
(* read system timer *)
tx := DWORD_TO_TIME(T_PLC_MS());

ESR_Flag := FALSE;
esr_out[3].typ := 0;
esr_out[2].typ := 0;
esr_out[1].typ := 0;
esr_out[0].typ := 0;
cnt := 0;

(* check if inputs have chaged and fill buffer *)
IF s0 <> X0 AND ((s0 < 100) OR (S0 > 99 AND S0 < 200 AND mode >= 2) OR (S0 > 199 AND mode = 3)) THEN
	esr_out[cnt] := status_to_ESR(s0, a0, DT_in, TX);
	X0 := S0;
	cnt := cnt + 1;
	esr_flag := TRUE;
END_IF;
IF s1 <> X1 AND ((s1 < 100) OR (S1 > 99 AND S1 < 200 AND mode >= 2) OR (S1 > 199 AND mode = 3)) THEN
	esr_out[cnt] := status_to_ESR(s1, a1, DT_in, TX);
	X1 := S1;
	cnt := cnt + 1;
	esr_flag := TRUE;
END_IF;
IF s2 <> X2 AND ((s2 < 100) OR (S2 > 99 AND S2 < 200 AND mode >= 2) OR (S2 > 199 AND mode = 3)) THEN
	esr_out[cnt] := status_to_ESR(s2, a2, DT_in, TX);
	X2 := S2;
	cnt := cnt + 1;
	esr_flag := TRUE;
END_IF;
IF s3 <> X3 AND ((s3 < 100) OR (S3 > 99 AND S3 < 200 AND mode >= 2) OR (S3 > 199 AND mode = 3)) THEN
	esr_out[cnt] := status_to_ESR(s3, a3, DT_in, TX);
	X3 := S3;
	cnt := cnt + 1;
	esr_flag := TRUE;
END_IF;
IF cnt < 4 AND s4 <> X4 AND ((s4 < 100) OR (S4 > 99 AND S4 < 200 AND mode >= 2) OR (S4 > 199 AND mode = 3)) THEN
	esr_out[cnt] := status_to_ESR(s4, a4, DT_in, TX);
	X4 := S4;
	cnt := cnt + 1;
	esr_flag := TRUE;
END_IF;
IF cnt < 4 AND s5 <> X5 AND ((s5 < 100) OR (S5 > 99 AND S5 < 200 AND mode >= 2) OR (S5 > 199 AND mode = 3)) THEN
	esr_out[cnt] := status_to_ESR(s5, a5, DT_in, TX);
	X5 := S5;
	cnt := cnt + 1;
	esr_flag := TRUE;
END_IF;
IF cnt < 4 AND s6 <> X6 AND ((s6 < 100) OR (S6 > 99 AND S6 < 200 AND mode >= 2) OR (S6 > 199 AND mode = 3)) THEN
	esr_out[cnt] := status_to_ESR(s6, a6, DT_in, TX);
	X6 := S6;
	cnt := cnt + 1;
	esr_flag := TRUE;
END_IF;
IF cnt < 4 AND s7 <> X7 AND ((s7 < 100) OR (S7 > 99 AND S7 < 200 AND mode >= 2) OR (S7 > 199 AND mode = 3)) THEN
	esr_out[cnt] := status_to_ESR(s7, a7, DT_in, TX);
	X7 := S7;
	cnt := cnt + 1;
	esr_flag := TRUE;
END_IF;


(* revision history
hm	26. jan 2007		rev 1.0
	original version

hm	17. sep 2007	rev 1.1
	replaced time() with T_PLC_MS() for compatibility reasons
	
*)
END_FUNCTION_BLOCK

(* POU Other/status_to_ESR, ST *)
FUNCTION status_to_ESR : esr_data
VAR_INPUT
	status : BYTE;
	adress : STRING(10);
	DT_in : DT;
	TS : TIME;
END_VAR
VAR
END_VAR

(*
version 1.0	6 oct 2006
programmer 	hugo
tested by		tobias

status_to_esr creates esr data from a status byte.

*)
IF status < 100 THEN
	status_to_ESR.typ := 1;
ELSIF status < 200 THEN
	status_to_ESR.typ := 2;
ELSE
	status_to_ESR.typ := 3;
END_IF;
status_to_ESR.adress:= adress;
status_to_ESR.DS := DT_in;
status_to_ESR.TS := TS;
status_to_ESR.data[0] := status;
END_FUNCTION

(* POU Other/Oscat_version, ST *)
FUNCTION Oscat_version : DWORD
VAR_INPUT
	in : BOOL;
END_VAR
VAR
END_VAR


(*
version 1.1	16 dec 2007
programmer 	hugo
tested by		tobias

oscat_version returns the version number in dword format
132 is library version 1.32
if IN = true, the release date will be returned

*)
IF in THEN
	Oscat_version := DATE_TO_DWORD(D#2008-3-15);
ELSE
	Oscat_version := 272;
END_IF;

(* revision history
hm	6. oct 2006	rev 1.0
	original version

hm	16. dec 2007	rev 1.1
	added possibility to return date and version depending on IN.
 
*)
END_FUNCTION

(* POU String/BYTE_TO_STRB, ST *)
FUNCTION BYTE_TO_STRB : STRING
VAR_INPUT
	IN : BYTE;
END_VAR
VAR
	i: INT;
	pt : POINTER TO BYTE;
END_VAR

(*
version 1.1	15 dec 2007
programmer 	hugo
tested by		tobias

BYTE_TO_STRINGB converts a Byte to a String of Bits represented by '0' and '1' s.
The lowest order bit will be on the right and the high order bit on the left.

*)
(* pointer für die ausgabe ermitteln *)
pt := ADR(BYTE_TO_STRB);
(* die 8 ausgabecharacter ermitteln und schreiben *)
FOR i := 1 TO 8 DO
	IF in.7 THEN pt^ := 49; ELSE pt^ := 48; END_IF;
	in := SHL(in,1);
	pt := pt + 1;
END_FOR;

(* der ausgabestring muss noch mit 0 abgeschlossen werden *)
pt^ := 0;

(* code before rev 1.1
FOR i := 1 TO 8 DO
	IF in.0 = 0 THEN temp := CONCAT('0', temp); ELSE temp := CONCAT('1', temp); END_IF;
	in := SHR(in, 1);
END_FOR;
BYTE_TO_STRB := temp;
*)


(* revision history

hm		9.6.2007	rev 1.0		
	original version 

hm	15. dec 2007	rev 1.1
	inprooved code for higher performance

*)
END_FUNCTION

(* POU String/BYTE_TO_STRH, ST *)
FUNCTION BYTE_TO_STRH : STRING
VAR_INPUT
	IN : BYTE;
END_VAR
VAR
	temp : BYTE;
	PT : POINTER TO BYTE;
END_VAR

(*
version 1.2	15 dec 2007
programmer 	hugo
tested by		tobias

BYTE_TO_STRINGH converts a Byte to a String of Hexadecimal represented by '0' .. '9' and 'A' .. 'F'.
The lowest order Character will be on the right and the high order Character on the left.

*)
(* read pointer to output string *)
PT := ADR(BYTE_TO_STRH);
(* calculate high order hex value *)
temp := SHR(in,4);
(* convert value to hex character *)
IF temp <= 9 THEN temp := temp + 48; ELSE temp := temp + 55; END_IF;
(* write friat character to output string *)
PT^ := temp;
(* calculate low order hex value *)
temp := in AND 2#00001111;
IF temp <= 9 THEN temp := temp + 48; ELSE temp := temp + 55; END_IF;
(* increment pointer and wirte low order character *)
pt := pt + 1;
pt^ := temp;
(* set pointer at the end of the output string and close the string with 0 *)
pt := pt + 1;
pt^:= 0;


(* code before rev 1.2
FOR i := 1 TO 2 DO
	X := in AND 2#1111;
	IF X <= 9 THEN X := X + 48; ELSE X := X + 55; END_IF;
	Cx := CHR(X);
	temp := CONCAT(Cx, temp);
	in := SHR(in,4);
END_FOR;
BYTE_TO_STRH := temp;
*)

(* revision history

hm		9.6.2007		rev 1.0		
	original version 

hm		11.9.2007		rev 1.1		
	changed coding for compatibility with twincat, under twincat concat cannot have a function as argument.	

hm		15 dec 2007		REV 1.2
	changed code for higher performance
*)
END_FUNCTION

(* POU String/CAPITALIZE, ST *)
FUNCTION CAPITALIZE : STRING
VAR_INPUT
	str : STRING;
END_VAR
VAR
	PT : POINTER TO BYTE;
	pos : INT;
	L : INT;
	first : BOOL := TRUE;
END_VAR

(*
version 1.0	4. mar 2008
programmer 	hugo
tested by		tobias

uppercase returns str while all letters a..z and ä,ö,ü are converted to uppercase

*)
PT := ADR(CAPITALIZE);
CAPITALIZE := str;
L := LEN(str);
FOR pos := 1 TO l DO
	IF first THEN
		pt^ := TO_UPPER(pt^);
	END_IF;
	(* remember in first if the next char needs to capitalized *)
	IF pt^ = 32 THEN first := TRUE; ELSE first := FALSE; END_IF;
	PT := pt + 1;
END_FOR;

(* revision histroy
hm		4. mar 2008	rev 1.0
	original release

*)	
END_FUNCTION

(* POU String/TO_UPPER, ST *)
FUNCTION TO_UPPER : BYTE
VAR_INPUT
	IN : BYTE;
END_VAR
VAR
END_VAR

(*
version 1.0	6 mar 2008
programmer 	hugo
tested by		tobias

to_upper converts a character from lowercase to uppercase

*)
IF extended_ascii THEN
	IF ((in > 96) AND (in < 123)) OR ((in > 223) AND (in <> 247) AND (in <> 255)) THEN
		TO_UPPER := in AND 16#DF;
	ELSE
		TO_UPPER := in;
	END_IF;
ELSE
	IF ((in > 96) AND (in < 123)) THEN
		TO_UPPER := in AND 16#DF;
	ELSE
		TO_UPPER := in;
	END_IF;
END_IF;

(* revision history
hm		6. mar 2008	rev 1.0
	original version

*)
END_FUNCTION

(* POU String/DWORD_TO_STRB, ST *)
FUNCTION DWORD_TO_STRB : STRING
VAR_INPUT
	IN : DWORD;
END_VAR
VAR
	pt : POINTER TO BYTE;
	i: INT;
END_VAR

(*
version 1.1	15 dec 2007
programmer 	hugo
tested by		tobias

DWORD_TO_STRINGB converts a DWORD to a String of Bits represented by '0' and '1' s.
The lowest order bit will be on the right and the high order bit on the left.

*)
(* pointer für die ausgabe ermitteln *)
pt := ADR(DWORD_TO_STRB);
(* die 8 ausgabecharacter ermitteln und schreiben *)
FOR i := 1 TO 32 DO
	IF in.31 THEN pt^ := 49; ELSE pt^ := 48; END_IF;
	in := SHL(in,1);
	pt := pt + 1;
END_FOR;

(* der ausgabestring muss nochg mit 0 abgeschlossen werden *)
pt^ := 0;

(* revision history
hm		9.6.2007	rev 1.0		
	original version 
hm		15.dec 2007	rev 1.1
	changed code for better performance
*)
END_FUNCTION

(* POU String/DWORD_TO_STRF, ST *)
FUNCTION DWORD_TO_STRF : STRING
VAR_INPUT
	IN : DWORD;
	N : INT;
END_VAR
VAR
	L: INT;
	temp: STRING;
END_VAR

(*
version 1.0	26 jan 2007
programmer 	hugo
tested by		tobias

dword_to_strF converts a DWORD, BYTE or Word to a fixed length String.
the string will be filled with leading zeroes to achieve the fixed length, or if too long, the lowest digits will be used.

for example:	dword_to_strf(123,4) = '0123' 
				dword_to_strf(123,2) = '23'
*)
(* convert dword to string first and cut to length N *)
temp := RIGHT(DWORD_TO_STRING(in),N);
L := LEN(temp);
WHILE L < N DO
	temp := CONCAT('0', temp);
	L := L + 1;
END_WHILE;
DWORD_To_STRF := temp;
END_FUNCTION

(* POU String/DWORD_TO_STRH, ST *)
FUNCTION DWORD_TO_STRH : STRING
VAR_INPUT
	IN : DWORD;
END_VAR
VAR
	i : INT;
	temp : BYTE;
	pt : POINTER TO BYTE;
END_VAR

(*
version 1.2	15 dec 2007
programmer 	hugo
tested by		tobias

DWORD_TO_STRINGH converts a DWORD to a String of Hexadecimal represented by '0' .. '9' and 'A' .. 'F'.
The lowest order Character will be on the right and the high order Character on the left.

*)
(* read output adress to pointer *)
pt := ADR(DWORD_TO_STRH) + 8;
(* wirte the closing byte for the string *)
pt^:= 0;

(* write the 8 hex characters backwards *)
FOR i := 1 TO 8 DO;
	(* decrement the pointer *)
	pt := pt - 1;
	(* read the lowest order hex value *)
	temp := DWORD_TO_BYTE(in AND 16#0000000F);
	(* convert value to hex character *)
	IF temp <= 9 THEN temp := temp + 48; ELSE temp := temp + 55; END_IF;
	(* write character to output string *)
	PT^ := temp;
	(* shift in for nect hex character *)
	in := SHR(in,4);
END_FOR;


(* code beofre rev 1.2
FOR i := 1 TO 8 DO
	X := DWORD_TO_BYTE(in AND 2#1111);
	IF X <= 9 THEN X := X + 48; ELSE X := X + 55; END_IF;
	Cx := CHR(X);
	temp := CONCAT(Cx, temp);
	in := SHR(in,4);
END_FOR;
DWORD_TO_STRH := temp;
*)


(* revision history
hm		9.6.2007		rev 1.0		
	original version 

hm		11.9.2007		rev 1.1
	changed coding for compatibility with twincat, concat cannot support a function as an argument.

hm		15.12.2007		rev 1.2
	changed code for better performance
*)
END_FUNCTION

(* POU String/EXEC, ST *)
FUNCTION EXEC : STRING
VAR_INPUT
	str : STRING;
END_VAR
VAR
	pos: INT;
	R1: REAL;
	R2: REAL;
	operator: STRING;
END_VAR

(*
version 1.2	5. mar. 2008
programmer 	hugo
tested by		tobias

exec executes a mathematical term and returns the result as a string
the term can only be a simple term without brackets and only one operator
allowed operastors are: (+, -, *, /, ^, sqrt, sin, cos, tan).

*)
(* extract both numbers and operator *)
EXEC := UPPERCASE(TRIM(str));

pos := FINDB_NONUM(EXEC);
IF pos > 1 THEN R1 := STRING_TO_REAL(exec); END_IF;
R2 := STRING_TO_REAL(RIGHT(exec,LEN(exec)-pos));
exec := LEFT(exec,pos);
pos := findB_Num(exec);
operator := RIGHT(exec,LEN(exec) - pos);
IF operator = '' AND LEN(str) = 0 THEN
	exec := '';
	RETURN;
ELSIF operator = '' THEN
	exec := str;
	RETURN;
END_IF;
IF operator = '^' THEN
	exec := REAL_TO_STRING(EXPT(R1, R2));
ELSIF operator = 'SQRT' THEN
	exec := REAL_TO_STRING(SQRT(R2));
ELSIF operator = 'SIN' THEN
	EXEC := REAL_TO_STRING(SIN(r2));
ELSIF operator = 'COS' THEN
	exec := REAL_TO_STRING(COS(r2));
ELSIF operator = 'TAN' THEN
	exec := REAL_TO_STRING(TAN(R2));
ELSIF operator = '*' THEN
	exec := REAL_TO_STRING(R1 * R2);
ELSIF operator = '/' THEN
	IF R2 <> 0 THEN exec := REAL_TO_STRING(R1 / R2); ELSE exec := 'ERROR'; END_IF;
ELSIF operator = '+' THEN
	exec := REAL_TO_STRING(r1 + r2);
ELSIF operator = '-' THEN
	exec := REAL_TO_STRING(r1 - r2);
ELSE
	exec := 'ERROR';
END_IF;

(* some systems deliver n. instead of n.0 ! *)
IF RIGHT(EXEC,1) = '.' THEN EXEC := CONCAT(EXEC,'0'); END_IF;



(* revision history

hm 	6.feb 2007		rev 1.1
	cos has to be written in uppercase
	divide by 0 will return an error

hm		5. mar. 2008	rev 1.2
	add a 0 to the string if a '.' is at the end of the string     
*)
END_FUNCTION

(* POU String/UPPERCASE, ST *)
FUNCTION UPPERCASE : STRING
VAR_INPUT
	str : STRING;
END_VAR
VAR
	PT : POINTER TO BYTE;
	pos: INT;
	l: INT;
END_VAR

(*
version 1.1	4. feb 2008
programmer 	hugo
tested by		tobias

uppercase returns str while all letters a..z and ä,ö,ü are converted to uppercase

*)
PT := ADR(UPPERCASE);
uppercase := str;
l := LEN(str);
FOR pos := 1 TO l DO
	pt^ := TO_UPPER(pt^);
	PT := PT + 1;
END_FOR;

(* revision histroy
hm		6.10.2006		rev 1.0
	original release

hm		4. feb. 2008	rev 1.1
	improved performance
	added Ä,Ö,Ü

hm		6. mar 2008	rev 1.2
	added support for exteded Ascii
*)	
END_FUNCTION

(* POU String/TRIM, ST *)
FUNCTION TRIM : STRING
VAR_INPUT
	str : STRING;
END_VAR
VAR
	pos: INT;
END_VAR

(*
version 1.0	6 oct 2006
programmer 	hugo
tested by		tobias

the function deletes all blanks within a string.

*)
TRIM := str;
REPEAT
	pos := FIND(trim,' ');
	trim := REPLACE(trim,'',1,pos);
UNTIL pos = 0	END_REPEAT;


(* revision histroy
hm		6.10.2006		rev 1.0
	original release

*)
END_FUNCTION

(* POU String/FINDB_NONUM, ST *)
FUNCTION FINDB_NONUM : INT
VAR_INPUT
	str : STRING;
END_VAR
VAR
	pos: INT;
	pt : POINTER TO BYTE;
END_VAR

(*
version 1.1	29. feb 2008
programmer 	hugo
tested by		tobias

findB_noNum searches str backwards and returns the last position which is not a number.
a number is characterized by a letter "0..9" or "."

*)
pt := ADR(str) + LEN(str) - 1;
FOR pos := LEN(str) TO 1 BY -1 DO;
	IF NOT((PT^ > 47 AND PT^ < 58) OR PT^ = 46) THEN
		FINDB_NONUM := pos;
		RETURN;
	END_IF;
	PT := PT - 1;
END_FOR;
FINDB_NONUM := 0;


(* revision history
hm		6. oct 2006	rev 1.0
	original version

hm		29. feb 2008	rev 1.1
	improved performance
*)
END_FUNCTION

(* POU String/FINDB_NUM, ST *)
FUNCTION FINDB_NUM : INT
VAR_INPUT
	str : STRING;
END_VAR
VAR
	pos: INT;
	pt : POINTER TO BYTE;
END_VAR

(*
version 1.1	29. feb 2008
programmer 	hugo
tested by		tobias

findB_Num searches str backward and returns the last position of a number
a number is characterized by a letter "0..9" or "."

*)
pt := ADR(str) + LEN(str) - 1;
FOR pos := LEN(str) TO 1 BY -1 DO;
	IF (PT^ > 47 AND PT^ < 58) OR PT^ = 46 THEN
		FINDB_NUM := pos;
		RETURN;
	END_IF;
	PT := PT - 1;
END_FOR;
FINDB_NUM := 0;

(* revision history
hm		6. oct 2006	rev 1.0
	original version

hm		29. feb 2008	rev 1.1
	improved performance
*)
END_FUNCTION

(* POU String/FIND_CHAR, ST *)
FUNCTION FIND_CHAR : INT
VAR_INPUT
	str : STRING;
	pos : INT;
END_VAR
VAR
	i: INT;
	pt : POINTER TO ARRAY[1..255] OF BYTE;
	stop: INT;
	X: BYTE;
END_VAR

(*
version 1.0	29. feb 2008
programmer 	hugo
tested by		tobias

find_char searches str and returns the starting position of the first character that is not a control character.
control characters are the ascii character 00 .. 31.

*)
pt := ADR(str);
stop := LEN(str);
FOR i := MAX(pos,1) TO stop DO;
	X := pt^[i];
	IF X > 31 THEN
		FIND_CHAR := i;
		RETURN;
	END_IF;
END_FOR;
FIND_CHAR := 0;


(* revision history
hm		29. feb 2008	rev 1.0
	original version

*)
END_FUNCTION

(* POU String/FIND_CTRL, ST *)
FUNCTION FIND_CTRL : INT
VAR_INPUT
	str : STRING;
	pos : INT;
END_VAR
VAR
	i: INT;
	pt : POINTER TO ARRAY[1..255] OF BYTE;
	stop: INT;
	x: BYTE;
END_VAR

(*
version 1.0	29. feb 2008
programmer 	hugo
tested by		tobias

find_ctrl searches str and returns the starting position of a control character
control characters are the ascii character 00 .. 31.

*)
pt := ADR(str);
stop := LEN(str);
FOR i := MAX(pos,1) TO stop DO;
	x := PT^[I];
	IF x < 32 THEN
		FIND_CTRL := i;
		RETURN;
	END_IF;
END_FOR;
FIND_CTRL := 0;


(* revision history
hm		29. feb 2008	rev 1.0
	original version

*)
END_FUNCTION

(* POU String/FIND_NONUM, ST *)
FUNCTION FIND_NONUM : INT
VAR_INPUT
	str : STRING;
	pos : INT;
END_VAR
VAR
	i: INT;
	pt : POINTER TO ARRAY[1..255] OF BYTE;
	end: INT;
	X: BYTE;
END_VAR

(*
version 1.1	29. feb 2008
programmer 	hugo
tested by		tobias

find_noNum searches str and returns the first position which is not a number.
a number is characterized by a letter "0..9" or "."

*)
pt := ADR(str);
end := LEN(str);
FOR i := MAX(pos,1) TO end DO;
	X := pt^[i];
	IF NOT((X > 47 AND X < 58) OR X = 46) THEN
		FIND_NONUM := i;
		RETURN;
	END_IF;
END_FOR;
FIND_NONUM := 0;


(* revision history
hm		6. oct. 2006	rev 1.0
	original version

hm		29. feb 2008	rev 1.1
	added input pos to start search at position

*)
END_FUNCTION

(* POU String/FIND_NUM, ST *)
FUNCTION FIND_NUM : INT
VAR_INPUT
	str : STRING;
	pos : INT;
END_VAR
VAR
	i : INT;
	pt : POINTER TO ARRAY[1..255] OF BYTE;
	stop : INT;
	X: BYTE;
END_VAR

(*
version 1.1	29. feb 2008
programmer 	hugo
tested by		tobias

find_Num searches str and returns the starting position of a number
a number is characterized by a letter "0..9" or "."

*)
pt := ADR(str);
stop := LEN(str);
FOR i := MAX(pos,1) TO stop DO;
	X := pt^[i];
	IF (X > 47 AND X < 58) OR X = 46 THEN
		FIND_NUM := i;
		RETURN;
	END_IF;
END_FOR;
FIND_NUM := 0;


(* revision history
hm		6. oct. 2006	rev 1.0
	original version

hm		29. feb 2008	rev 1.1
	added input pos to start search at position

*)
END_FUNCTION

(* POU String/FINDB, ST *)
FUNCTION FINDB : INT
VAR_INPUT
	str1 : STRING;
	str2 : STRING;
END_VAR
VAR
	pos: INT;
	length: INT;
END_VAR

(*
version 1.2	29. feb 2008
programmer 	hugo
tested by		tobias

the function find searches an str1 for the presence of str2 and returns the first position of str1 of the last presence in instring.
the function is similar to find except it searches from the right to left.
 a 0 is returned if the string is not found.

